  rq_init_comm_if_connected(9, "1")
  rq_init_comm_if_connected(2, "2")
  rq_init_comm_if_connected(3, "3")
  rq_init_comm_if_connected(4, "4")
  rq_print_connected_grippers()
  rq_gripper_communication_thread = run rq_gripper_communication()
  set_closed_norm(100.0, 1)
  set_open_norm(0.0, 1)
  set_closed_mm(0.0, 1)
  set_open_mm(50.0, 1)
  set_closed_norm(89.80392156862744, 2)
  set_open_norm(1.1764705882352942, 2)
  set_closed_mm(0.0, 2)
  set_open_mm(85.0, 2)
  set_closed_norm(100.0, 3)
  set_open_norm(0.0, 3)
  set_closed_mm(0.0, 3)
  set_open_mm(50.0, 3)
  set_closed_norm(100.0, 4)
  set_open_norm(0.0, 4)
  set_closed_mm(0.0, 4)
  set_open_mm(50.0, 4)
  rq_current_limit_enabled = False
  while(not rq_gripper_communication_thread_started):
      sleep(0.008)
  end
  # end: URCap Installation Node
  step_count_4a6500cf_8076_4a8b_917a_8f51ecf751d7 = 0.0
  thread Step_Counter_Thread_413bcd2b_4cc3_4dfb_b837_23a851721193():
    while (True):
      step_count_4a6500cf_8076_4a8b_917a_8f51ecf751d7 = step_count_4a6500cf_8076_4a8b_917a_8f51ecf751d7 + 1.0
      sync()
    end
  end
  run Step_Counter_Thread_413bcd2b_4cc3_4dfb_b837_23a851721193()
  global Waypoint_2_p=p[.280607659900, -.116080070486, .398046390840, -2.237106331319, 2.146374778909, -.035913347281]
  global Waypoint_2_q=[0.051861584186553955, -1.5388997805169602, -1.1589003801345825, 4.315436525935791, 1.571950912475586, 0.011884484440088272]
  global Waypoint_64_p=p[.354470099489, -.115863572825, .377183440885, -3.127244589782, -.024157028155, -.017479675085]
  global Waypoint_64_q=[0.04108531400561333, -1.8477684460081996, -0.895115852355957, 4.326324625606201, 1.5751920938491821, -1.5445211569415491]
  global Waypoint_65_p=p[.360926107403, -.115109045274, .191361701352, -3.127293402598, -.024210541102, -.017289759710]
  global Waypoint_65_q=[0.04325436055660248, -1.9099999866881312, -1.7111023664474487, 5.204389768629827, 1.5756800174713135, -1.549448315297262]
  global Waypoint_66_p=p[.360932787725, -.115104634702, .343669410000, -3.127285727102, -.024216683853, -.017394975926]
  global Waypoint_66_q=[0.042698003351688385, -1.8273731670775355, -1.0869383811950684, 4.497707052821777, 1.5746601819992065, -1.5442584196673792]
  global Waypoint_67_p=p[.360931648608, -.115099983374, .343682798901, .037017771719, -3.130286849386, .022250894461]
  global Waypoint_67_q=[0.049796681851148605, -1.8348614178099574, -1.0676213502883911, 4.462740107173584, 1.5471274852752686, 1.5965529680252075]
  global Waypoint_68_p=p[.369452922664, -.269494866094, .114409751435, .034594999463, -2.558735015916, -1.790314713905]
  global Waypoint_68_q=[-0.506531063710348, -3.1360022030272425, 0.2904461065875452, 3.4742390352436523, 2.5075576305389404, 0.5356799960136414]
  global Waypoint_79_p=p[.369461792411, -.269489790217, .091378168109, .034671000925, -2.558784123149, -1.790337845898]
  global Waypoint_79_q=[-0.5066073576556605, -3.2201863727965296, 0.36221200624574834, 3.4865333276936035, 2.507685422897339, 0.5354438424110413]
  global Waypoint_73_p=p[.355312960958, -.120113755208, .193383739669, -2.219409439704, 2.165038969222, -.036333231459]
  global Waypoint_73_q=[0.030303990468382835, -1.8856717548766078, -1.7507002353668213, 5.25380157211379, 1.5736638307571411, -0.0011132399188440445]
  global Waypoint_77_p=p[.355960533253, -.120111757755, .194005001047, -3.095268771574, .046175877951, .006344872093]
  global Waypoint_77_q=[0.02114737220108509, -1.8991791210570277, -1.7065989971160889, 5.174873578339376, 1.6078295707702637, -1.5260933081256312]
  global Waypoint_70_p=p[.369313361026, -.121750279780, .239195417816, .036983595410, -3.130201769342, .022288106508]
  global Waypoint_70_q=[0.030927900224924088, -1.8825870953001917, -1.4988759756088257, 4.941975313216009, 1.5469911098480225, 1.5737316608428955]
  global Waypoint_71_p=p[.355771906615, -.117714048296, .191403478305, -2.239338673519, 2.148294993320, -.040719651885]
  global Waypoint_71_q=[0.03811154514551163, -1.8879105053343714, -1.758138656616211, 5.26347969749526, 1.5698184967041016, -0.010163132344381154]
  global Waypoint_72_p=p[.361680845210, -.117399576394, .187815914645, -3.134574229139, .018986447884, .007833898805]
  global Waypoint_72_q=[0.038440003991127014, -1.9243623218932093, -1.7018784284591675, 5.193334001093664, 1.569042444229126, -1.5266807715045374]
  global Waypoint_75_p=p[.361669157885, -.117405189295, .336567976331, -3.134554026129, .018916398175, .007773225074]
  global Waypoint_75_q=[0.03786372393369675, -1.8343554935851039, -1.105195164680481, 4.50668923437085, 1.5680339336395264, -1.5216921011554163]
  global Waypoint_76_p=p[.369461443324, -.267242268416, .139990265830, -1.905707976787, .019547548118, .054785252250]
  global Waypoint_76_q=[-0.5030587355243128, -2.9809848270811976, 0.07564908662904912, 3.5141541200825195, 2.516566038131714, -2.5729287306415003]
  global Waypoint_78_p=p[.363433709975, -.271007124876, .085521034428, -1.833243928261, .011816409372, .027475621175]
  global Waypoint_78_q=[-0.5206573645221155, -3.1302629909911097, 0.13170367876161748, 3.4938294130512695, 2.5485825538635254, -2.691174332295553]
  global Waypoint_74_p=p[.354955148094, -.112489845695, .193442052840, -.170335331910, 3.121840961438, -.070471601362]
  global Waypoint_74_q=[0.06705623120069504, -1.8727036915221156, -1.7540733814239502, 5.212656187802114, 1.5166053771972656, 1.5219447612762451]
  global Waypoint_8_p=p[.360358944520, -.116083441389, .194376541524, -2.248047450183, 2.157812796511, .002217808263]
  global Waypoint_8_q=[0.039292335510253906, -1.9029251537718714, -1.7079429626464844, 5.199970382242956, 1.5806336402893066, -0.007966343556539357]
  global Waypoint_11_p=p[.360346612111, -.116074708299, .194372829697, -.134360355414, 3.119145978590, -.025737827061]
  global Waypoint_11_q=[0.048485033214092255, -1.8981090984740199, -1.7157262563705444, 5.205127703934469, 1.5453232526779175, 1.5264861583709717]
  global Waypoint_13_p=p[.360128512254, -.115917649696, .194944831011, -2.245984467664, 2.155060370290, -.017546589543]
  global Waypoint_13_q=[0.041585683822631836, -1.8980418644347132, -1.716995120048523, 5.215424525528707, 1.5738275051116943, -0.006153885518209279]
  global Waypoint_12_p=p[.360146406837, -.115908484738, .194960409380, -3.112369099282, -.068557507067, .019286775543]
  global Waypoint_12_q=[0.03719525411725044, -1.907412668267721, -1.6854465007781982, 5.152547257929601, 1.5902478694915771, -1.583886448537008]
  global Waypoint_14_p=p[.365368782725, -.113055548392, .194065158575, -2.254756102503, 2.163756251815, .001000413874]
  global Waypoint_14_q=[0.048927538096904755, -1.9188252888121546, -1.6842378377914429, 5.186415302544393, 1.5737271308898926, 0.0014259815216064453]
  global Waypoint_15_p=p[.365366593966, -.113055726856, .313338506786, -2.254649094383, 2.163740256071, .001003954948]
  global Waypoint_15_q=[0.04848504066467285, -1.8237744770445765, -1.2354748249053955, 4.642688437099121, 1.572627305984497, 0.005483102984726429]
  global Waypoint_23_p=p[.365372287050, -.113060920253, .392746291245, -3.129916090772, .002408869415, .018908326558]
  global Waypoint_23_q=[0.04779151454567909, -1.957900186578268, -0.647434651851654, 4.165631933803223, 1.5744084119796753, -1.519916836415426]
  global Waypoint_16_p=p[.363125696366, -.264930337535, .106644692126, -1.930464727729, -.006616513493, -.014136172145]
  global Waypoint_16_q=[-0.5062182585345667, -2.7471419773497523, -0.5786928534507751, 3.9979278284260253, 2.5275027751922607, -2.5754240194903772]
  global Waypoint_17_p=p[.359006490406, -.116088333119, .193010890574, -2.237057782096, 2.146370407089, -.035922785381]
  global Waypoint_17_q=[0.041281212121248245, -1.8952018223204554, -1.7393155097961426, 5.252011346607961, 1.5739600658416748, -0.00670034090151006]
  global Waypoint_18_p=p[.359004234930, -.116091493614, .368940192177, -2.237123790240, 2.146381621509, -.035885413675]
  global Waypoint_18_q=[0.04060101509094238, -1.8347741566100062, -0.9686561226844788, 4.42090289175, 1.5729669332504272, -7.427374469202164E-4]
  global Waypoint_19_p=p[.359011315786, -.116090988468, .368946186542, -3.094932517113, -.087303060908, .020290804464]
  global Waypoint_19_q=[0.031704679131507874, -1.8744904003539027, -0.8905159831047058, 4.323864622707031, 1.6067882776260376, -1.5951746145831507]
  global Waypoint_20_p=p[.366236911694, -.120423048900, .235895888638, -3.094888190076, -.087401744852, .020371246681]
  global Waypoint_20_q=[0.01979127898812294, -1.8803430996336878, -1.5173594951629639, 4.955764177232542, 1.6063188314437866, -1.6122682730304163]
  global Waypoint_21_p=p[.364127453615, -.117777467803, .193292956992, -2.256931465612, 2.166078680800, .016499453347]
  global Waypoint_21_q=[0.03465377166867256, -1.9235106907286585, -1.6773513555526733, 5.174797373801031, 1.5786932706832886, -0.01269084612001592]
  global Waypoint_32_p=p[.364117039848, -.117791711540, .193288967422, -.001509992748, 3.124739503024, -.003616906989]
  global Waypoint_32_q=[0.03972397744655609, -1.9184686146178187, -1.6911675930023193, 5.198225903301992, 1.558967113494873, 1.6030347347259521]
  global Waypoint_24_p=p[.356858385198, -.114748285525, .193459227445, -2.236998775234, 2.146447506006, -.035874401211]
  global Waypoint_24_q=[0.045367274433374405, -1.8846894703307093, -1.7517141103744507, 5.253918099194326, 1.5737637281417847, -0.0025556723224084976]
  global Waypoint_25_p=p[.356855401252, -.114737739719, .388234546256, -2.237156328648, 2.146401722995, -.035868096178]
  global Waypoint_25_q=[0.04460291564464569, -1.8599993191161097, -0.837320864200592, 4.314809961909912, 1.5731350183486938, 0.004033051431179047]
  global Waypoint_27_p=p[.356862717244, -.114749303796, .388207810464, -3.101225685288, -.061188193992, .021131354318]
  global Waypoint_27_q=[0.0369672067463398, -1.9050165615477503, -0.7486847043037415, 4.212594671840332, 1.6017820835113525, -1.5721553007708948]
  global Waypoint_26_p=p[.365655111079, -.272422037322, .090212739427, -1.849444862553, -.046251879190, -.014050237907]
  global Waypoint_26_q=[-0.519848648701803, -3.0603820286192835, 0.005677525197164357, 3.5761772829243164, 2.5399975776672363, -2.73091704050173]
  global Waypoint_28_p=p[.354352026237, -.116082337067, .201505476102, -2.237022096588, 2.146441145418, -.035930660985]
  global Waypoint_28_q=[0.04179730266332626, -1.861342569390768, -1.741385579109192, 5.2202181098754785, 1.573683500289917, -0.005864922200338185]
  global Waypoint_29_p=p[.354342109747, -.116082273200, .351046674865, -2.237104102966, 2.146365455752, -.035900070297]
  global Waypoint_29_q=[0.04126540571451187, -1.7894679508604945, -1.1141570806503296, 4.521125956172607, 1.5726195573806763, -8.066336261194351E-4]
  global Waypoint_30_p=p[.354353116406, -.116080119546, .351018725794, -3.094806654881, -.093017323019, .020491730000]
  global Waypoint_30_q=[0.032280921936035156, -1.824392934838766, -1.0455470085144043, 4.428581400508545, 1.6063028573989868, -1.5990260283099573]
  global Waypoint_31_p=p[.368984100378, -.120915937945, .229682487256, -3.095748275296, .014195489245, .018015526971]
  global Waypoint_31_q=[0.018162259832024574, -1.8980938396849574, -1.5245105028152466, 4.9836007235343835, 1.6071596145629883, -1.5484493414508265]
  global Waypoint_22_p=p[.364116883869, -.117782716197, .193288229298, -3.139205010194, -.012449845557, .026525647038]
  global Waypoint_22_q=[0.03819990158081055, -1.9253126583495082, -1.6663216352462769, 5.146627026587286, 1.5645008087158203, -1.5466154257403772]
  global Waypoint_33_p=p[.365384650811, -.113046739845, .368046327177, -.082065141775, 3.127997038214, -.017202640169]
  global Waypoint_33_q=[0.05418265983462334, -1.8752075634398402, -0.9042851328849792, 4.363438292140625, 1.5500004291534424, 1.5726572275161743]
  global Waypoint_34_p=p[.363742157567, -.276249559590, .088704299793, -.017752167727, 2.507683090614, 1.878743902822]
  global Waypoint_34_q=[-0.5293481985675257, -3.0111896000304164, -0.10669158399105072, 3.651848478908203, 2.5413897037506104, 0.4435216784477234]
  global Waypoint_35_p=p[.365353984843, -.113065797339, .314962777279, -3.129998929491, -.008745881210, .018959456628]
  global Waypoint_35_q=[0.04835740104317665, -1.834442754785055, -1.204733967781067, 4.599378271693848, 1.5727750062942505, -1.5296428839312952]
  global Waypoint_36_p=p[.365363249284, -.113054207165, .238209290372, -3.129975666367, -.008814066519, .018790901880]
  global Waypoint_36_q=[0.04866836220026016, -1.8599559269347132, -1.5340592861175537, 4.954310434847631, 1.573059320449829, -1.532309357319967]
  global Waypoint_37_p=p[.365360195551, -.113055658309, .193805528531, -3.129976498904, -.008769838028, .018833791209]
  global Waypoint_37_q=[0.04882422462105751, -1.923554082910055, -1.6685000658035278, 5.152311789780416, 1.573791742324829, -1.5337484518634241]
  global Waypoint_38_p=p[.364249601416, -.113557103657, .190832473293, 2.204318959610, 2.224300240519, -.048856099106]
  global Waypoint_38_q=[0.05790204554796219, -1.921460290948385, -1.6850007772445679, 5.161710727005758, 1.5336676836013794, -3.0986831823932093]
  global Waypoint_39_p=p[.364266614325, -.110421946332, .190856746275, 2.209420651831, 2.229591677071, -.037414170316]
  global Waypoint_39_q=[0.06399016082286835, -1.9190217457213343, -1.6884911060333252, 5.163263070374288, 1.544034719467163, -3.092748228703634]
  global Waypoint_40_p=p[.364268983895, -.110435285300, .361886964377, 2.209420466399, 2.229618306717, -.037429530523]
  global Waypoint_40_q=[0.06325225532054901, -1.8707810841002406, -0.9290131330490112, 4.355386896724365, 1.5435824394226074, -3.086977783833639]
  global Waypoint_41_p=p[.364265840443, -.110427102269, .361870025237, -3.125110448973, -.105776433446, .029932400516]
  global Waypoint_41_q=[0.05484846606850624, -1.8776551685728968, -0.9186587929725647, 4.349270983333252, 1.5762443542480469, -1.5833638350116175]
  global Waypoint_42_p=p[.369042632900, -.110424594122, .224326920210, -3.126301319343, -.005632380127, .029185961145]
  global Waypoint_42_q=[0.05444587022066116, -1.889749666253561, -1.5589039325714111, 5.0025426028068445, 1.5772563219070435, -1.5249899069415491]
  global Waypoint_43_p=p[.365353936489, -.113064268181, .322294641646, -2.254796238667, 2.163800975117, .001120761204]
  global Waypoint_43_q=[0.04843675345182419, -1.8276883564391078, -1.1881848573684692, 4.59915463506665, 1.5726237297058105, 0.0057464404962956905]
  global Waypoint_44_p=p[.365369713945, -.113043464009, .322292976272, -3.129186148249, -.086620865562, .019272676305]
  global Waypoint_44_q=[0.04855327680706978, -1.8383614025511683, -1.1648505926132202, 4.562915487880371, 1.5721629858016968, -1.5789158979998987]
  global Waypoint_45_p=p[.365392044628, -.271165795022, .097080861471, -1.854532438468, -.060032954149, -.026643104538]
  global Waypoint_45_q=[-0.5176385084735315, -2.9681459865965785, -0.158863827586174, 3.659778280849121, 2.540245294570923, -2.7370362917529505]
  global Waypoint_46_p=p[.365359176267, -.113063290570, .333428241271, -2.254692977086, 2.163738544463, .000970293766]
  global Waypoint_46_q=[0.04838533699512482, -1.8350216350951136, -1.1259797811508179, 4.544436617488525, 1.5727194547653198, 0.006145970430225134]
  global Waypoint_47_p=p[.365371307895, -.113054913652, .333395021784, -3.130121874518, -.066020013586, .019874548846]
  global Waypoint_47_q=[0.048556797206401825, -1.8465644321837367, -1.1012637615203857, 4.507215185756348, 1.5719189643859863, -1.565303150807516]
  global Waypoint_48_p=p[.365368433594, -.110775889601, .232224413161, -3.130138965271, -.066016593977, .019854438479]
  global Waypoint_48_q=[0.0552668571472168, -1.8638464413084925, -1.5576152801513672, 4.98091487863616, 1.5721588134765625, -1.562469784413473]
  global Waypoint_52_p=p[.365359843959, -.113081349965, .194064897071, -3.129642378612, -.064303807651, .019061278977]
  global Waypoint_52_q=[0.04888356477022171, -1.9231182537474574, -1.667611002922058, 5.150625216751852, 1.5732671022415161, -1.5691588560687464]
  global Waypoint_49_p=p[.365357344058, -.113073281521, .368518599816, -3.129675426161, -.064295774517, .019011934194]
  global Waypoint_49_q=[0.04817046970129013, -1.8945962391295375, -0.8649749755859375, 4.319530649776123, 1.5729867219924927, -1.5631969610797327]
  global Waypoint_50_p=p[.371009155844, -.266422439514, .106051816126, -1.904984487247, -.030855415702, .036523254658]
  global Waypoint_50_q=[-0.49856454530824834, -2.904177804986471, -0.24639520049095154, 3.7509915071674804, 2.5077571868896484, -2.622943703328268]
  global Waypoint_51_p=p[.365365756281, -.113068067212, .335109436071, -2.254715734372, 2.163808014871, .001013615422]
  global Waypoint_51_q=[0.048369091004133224, -1.8364578686156214, -1.116073727607727, 4.535901232356689, 1.5727112293243408, 0.0062180995009839535]
  global Waypoint_53_p=p[.363190347376, -.109909249167, .214454177245, 2.202648627526, 2.239361144151, -.026164233321]
  global Waypoint_53_q=[0.0639103502035141, -1.8745748005309046, -1.631171464920044, 5.0654775378997705, 1.5498764514923096, -3.099539581929342]
  global Waypoint_54_p=p[.365364617238, -.113046544047, .193803919468, -2.147317235435, 2.270276089319, -.000280218377]
  global Waypoint_54_q=[0.04924694821238518, -1.9189378223814906, -1.6859766244888306, 5.189448195486822, 1.572607398033142, 0.0985577404499054]
  global Waypoint_55_p=p[.369046237243, -.110420112971, .224327646614, -2.257586529246, 2.150383646731, .005568399145]
  global Waypoint_55_q=[0.05381538346409798, -1.8819652996458949, -1.5833349227905273, 5.051859217673101, 1.5802409648895264, 4.339217866800027E-6]
  global Waypoint_56_p=p[.364264927128, -.116054024615, .192333636877, -3.095046149511, .058807189831, .016907900219]
  global Waypoint_56_q=[0.03184909746050835, -1.929457803765768, -1.669385313987732, 5.161799806147375, 1.6082003116607666, -1.5073078314410608]
  global Waypoint_57_p=p[.364253565471, -.116069606295, .333900611097, -3.095734687662, -.040512408598, .019114780625]
  global Waypoint_57_q=[0.031436286866664886, -1.85087313274526, -1.0939775705337524, 4.505091353053711, 1.6066334247589111, -1.5665701071368616]
  global Waypoint_58_p=p[.365317983006, -.268384127780, .096470187856, -1.827396022314, -.032757791678, -.006341395965]
  global Waypoint_58_q=[-0.514263931904928, -3.06442989925527, 0.04053718248476201, 3.5144497591206054, 2.5557875633239746, -2.7419408003436487]
  global Waypoint_59_p=p[.361348202281, -.116091074418, .193171940183, -2.255348123474, 2.164443027209, .005235593744]
  global Waypoint_59_q=[0.04056864231824875, -1.9096676311888636, -1.7008389234542847, 5.191219466715612, 1.5751317739486694, -0.006904427205220998]
  global Waypoint_60_p=p[.361353719735, -.116078329177, .193164234402, -.107411230804, 3.126172424726, -.013320009558]
  global Waypoint_60_q=[0.04628801345825195, -1.906170507470602, -1.7079107761383057, 5.199406075268545, 1.553221583366394, 1.5418486595153809]
  global Waypoint_62_p=p[.357407157421, -.114500090328, .192443539627, -2.237115183190, 2.146339057492, -.035930597557]
  global Waypoint_62_q=[0.04602402448654175, -1.8884631596007289, -1.7518619298934937, 5.257864701538839, 1.5737314224243164, -0.0020354429828088882]
  global Waypoint_61_p=p[.357808555570, -.114512094935, .192817914002, -3.094022297870, -.120534455071, .014031671817]
  global Waypoint_61_q=[0.037067364901304245, -1.9025441608824671, -1.7050750255584717, 5.170009690314092, 1.6068851947784424, -1.6179912726031702]
  global Waypoint_63_p=p[.361345425225, -.116096314852, .193167637645, 2.081805564531, 2.284545736471, .059854815242]
  global Waypoint_63_q=[0.04617943987250328, -1.8987189731993617, -1.7417824268341064, 5.275271165161886, 1.5542293787002563, 3.087625741958618]
  $ 2 "Robot Program"
  $ 3 "Mouvements L'"
  $ 4 "MoveJ"
  $ 5 "Waypoint_2" "breakAfter"
  movej(get_inverse_kin(Waypoint_2_p, qnear=Waypoint_2_q), a=1.3962634015954636, v=1.0471975511965976)
  $ 6 "MoveJ"
  $ 7 "Waypoint_64" "breakAfter"
  movej(get_inverse_kin(Waypoint_64_p, qnear=Waypoint_64_q), a=1.3962634015954636, v=1.0471975511965976)
  $ 8 "MoveJ"
  $ 9 "Waypoint_65" "breakAfter"
  movej(get_inverse_kin(Waypoint_65_p, qnear=Waypoint_65_q), a=1.3962634015954636, v=1.0471975511965976)
  # begin: URCap Program Node
  #   Source: Robotiq_Grippers, 1.8.11.21258, Robotiq Inc.
  #   Type: Gripper
  $ 10 "Gripper Close (2)"
  if not(gripper_connected[1]):
    popup("Gripper 2 must be connected to run this program.", "No connection", False, True, True)
  end
  if not(rq_is_gripper_activated("2")):
    popup("Gripper 2 is not activated. Go to Installation tab > Gripper to activate it and run the program again.", "Not activated", False, True, True)
  end
  rq_set_pos_spd_for(255, 0, 0, "2")
  rq_wait_pos_spe_for_request(255, 0, 0, "2")
  rq_go_to("2")
  rq_wait("2")
  # end: URCap Program Node
  $ 11 "MoveJ"
  $ 12 "Waypoint_66" "breakAfter"
  movej(get_inverse_kin(Waypoint_66_p, qnear=Waypoint_66_q), a=1.3962634015954636, v=1.0471975511965976)
  $ 13 "MoveJ"
  $ 14 "Waypoint_67" "breakAfter"
  movej(get_inverse_kin(Waypoint_67_p, qnear=Waypoint_67_q), a=1.3962634015954636, v=1.0471975511965976)
  $ 15 "MoveJ"
  $ 16 "Waypoint_68" "breakAfter"
  movej(get_inverse_kin(Waypoint_68_p, qnear=Waypoint_68_q), a=1.3962634015954636, v=1.0471975511965976)
  $ 17 "MoveJ"
  $ 18 "Waypoint_79" "breakAfter"
  movej(get_inverse_kin(Waypoint_79_p, qnear=Waypoint_79_q), a=1.3962634015954636, v=1.0471975511965976)
  # begin: URCap Program Node
  #   Source: Robotiq_Grippers, 1.8.11.21258, Robotiq Inc.
  #   Type: Gripper
  $ 19 "Gripper Open (2)"
  if not(gripper_connected[1]):
    popup("Gripper 2 must be connected to run this program.", "No connection", False, True, True)
  end
  if not(rq_is_gripper_activated("2")):
    popup("Gripper 2 is not activated. Go to Installation tab > Gripper to activate it and run the program again.", "Not activated", False, True, True)
  end
  rq_set_pos_spd_for(0, 0, 0, "2")
  rq_wait_pos_spe_for_request(0, 0, 0, "2")
  rq_go_to("2")
  rq_wait("2")
  # end: URCap Program Node
  $ 20 "MoveJ"
  $ 21 "Waypoint_2" "breakAfter"
  movej(get_inverse_kin(Waypoint_2_p, qnear=Waypoint_2_q), a=1.3962634015954636, v=1.0471975511965976)
  $ 22 "MoveJ"
  $ 23 "MoveJ"
  $ 24 "MoveJ"
  $ 25 "MoveJ"
  $ 26 "MoveJ"
  $ 27 "MoveJ"
  $ 28 "Waypoint_73" "breakAfter"
  movej(get_inverse_kin(Waypoint_73_p, qnear=Waypoint_73_q), a=1.3962634015954636, v=1.0471975511965976)
  # begin: URCap Program Node
  #   Source: Robotiq_Grippers, 1.8.11.21258, Robotiq Inc.
  #   Type: Gripper
  $ 29 "Gripper Close (2)"
  if not(gripper_connected[1]):
    popup("Gripper 2 must be connected to run this program.", "No connection", False, True, True)
  end
  if not(rq_is_gripper_activated("2")):
    popup("Gripper 2 is not activated. Go to Installation tab > Gripper to activate it and run the program again.", "Not activated", False, True, True)
  end
  rq_set_pos_spd_for(255, 0, 0, "2")
  rq_wait_pos_spe_for_request(255, 0, 0, "2")
  rq_go_to("2")
  rq_wait("2")
  # end: URCap Program Node
  $ 30 "MoveJ"
  $ 31 "Waypoint_77" "breakAfter"
  movej(get_inverse_kin(Waypoint_77_p, qnear=Waypoint_77_q), a=1.3962634015954636, v=1.0471975511965976)
  # begin: URCap Program Node
  #   Source: Robotiq_Grippers, 1.8.11.21258, Robotiq Inc.
  #   Type: Gripper
  $ 32 "Gripper Open (2)"
  if not(gripper_connected[1]):
    popup("Gripper 2 must be connected to run this program.", "No connection", False, True, True)
  end
  if not(rq_is_gripper_activated("2")):
    popup("Gripper 2 is not activated. Go to Installation tab > Gripper to activate it and run the program again.", "Not activated", False, True, True)
  end
  rq_set_pos_spd_for(0, 0, 0, "2")
  rq_wait_pos_spe_for_request(0, 0, 0, "2")
  rq_go_to("2")
  rq_wait("2")
  # end: URCap Program Node
  $ 33 "MoveJ"
  $ 34 "Waypoint_2" "breakAfter"
  movej(get_inverse_kin(Waypoint_2_p, qnear=Waypoint_2_q), a=1.3962634015954636, v=1.0471975511965976)
  $ 35 "MoveJ"
  $ 36 "Waypoint_64" "breakAfter"
  movej(get_inverse_kin(Waypoint_64_p, qnear=Waypoint_64_q), a=1.3962634015954636, v=1.0471975511965976)
  $ 37 "MoveJ"
  $ 38 "Waypoint_65" "breakAfter"
  movej(get_inverse_kin(Waypoint_65_p, qnear=Waypoint_65_q), a=1.3962634015954636, v=1.0471975511965976)
  # begin: URCap Program Node
  #   Source: Robotiq_Grippers, 1.8.11.21258, Robotiq Inc.
  #   Type: Gripper
  $ 39 "Gripper Close (2)"
  if not(gripper_connected[1]):
    popup("Gripper 2 must be connected to run this program.", "No connection", False, True, True)
  end
  if not(rq_is_gripper_activated("2")):
    popup("Gripper 2 is not activated. Go to Installation tab > Gripper to activate it and run the program again.", "Not activated", False, True, True)
  end
  rq_set_pos_spd_for(255, 0, 0, "2")
  rq_wait_pos_spe_for_request(255, 0, 0, "2")
  rq_go_to("2")
  rq_wait("2")
  # end: URCap Program Node
  $ 40 "MoveJ"
  $ 41 "Waypoint_66" "breakAfter"
  movej(get_inverse_kin(Waypoint_66_p, qnear=Waypoint_66_q), a=1.3962634015954636, v=1.0471975511965976)
  $ 42 "MoveJ"
  $ 43 "Waypoint_67" "breakAfter"
  movej(get_inverse_kin(Waypoint_67_p, qnear=Waypoint_67_q), a=1.3962634015954636, v=1.0471975511965976)
  $ 44 "MoveJ"
  $ 45 "Waypoint_70" "breakAfter"
  movej(get_inverse_kin(Waypoint_70_p, qnear=Waypoint_70_q), a=1.3962634015954636, v=1.0471975511965976)
  # begin: URCap Program Node
  #   Source: Robotiq_Grippers, 1.8.11.21258, Robotiq Inc.
  #   Type: Gripper
  $ 46 "Gripper Open (2)"
  if not(gripper_connected[1]):
    popup("Gripper 2 must be connected to run this program.", "No connection", False, True, True)
  end
  if not(rq_is_gripper_activated("2")):
    popup("Gripper 2 is not activated. Go to Installation tab > Gripper to activate it and run the program again.", "Not activated", False, True, True)
  end
  rq_set_pos_spd_for(0, 0, 0, "2")
  rq_wait_pos_spe_for_request(0, 0, 0, "2")
  rq_go_to("2")
  rq_wait("2")
  # end: URCap Program Node
  $ 47 "MoveJ"
  $ 48 "Waypoint_2" "breakAfter"
  movej(get_inverse_kin(Waypoint_2_p, qnear=Waypoint_2_q), a=1.3962634015954636, v=1.0471975511965976)
  $ 49 "MoveJ"
  $ 50 "Waypoint_71" "breakAfter"
  movej(get_inverse_kin(Waypoint_71_p, qnear=Waypoint_71_q), a=1.3962634015954636, v=1.0471975511965976)
  # begin: URCap Program Node
  #   Source: Robotiq_Grippers, 1.8.11.21258, Robotiq Inc.
  #   Type: Gripper
  $ 51 "Gripper Close (2)"
  if not(gripper_connected[1]):
    popup("Gripper 2 must be connected to run this program.", "No connection", False, True, True)
  end
  if not(rq_is_gripper_activated("2")):
    popup("Gripper 2 is not activated. Go to Installation tab > Gripper to activate it and run the program again.", "Not activated", False, True, True)
  end
  rq_set_pos_spd_for(255, 0, 0, "2")
  rq_wait_pos_spe_for_request(255, 0, 0, "2")
  rq_go_to("2")
  rq_wait("2")
  # end: URCap Program Node
  # begin: URCap Program Node
  #   Source: Robotiq_Grippers, 1.8.11.21258, Robotiq Inc.
  #   Type: Gripper
  $ 52 "Gripper Open (2)"
  if not(gripper_connected[1]):
    popup("Gripper 2 must be connected to run this program.", "No connection", False, True, True)
  end
  if not(rq_is_gripper_activated("2")):
    popup("Gripper 2 is not activated. Go to Installation tab > Gripper to activate it and run the program again.", "Not activated", False, True, True)
  end
  rq_set_pos_spd_for(0, 0, 0, "2")
  rq_wait_pos_spe_for_request(0, 0, 0, "2")
  rq_go_to("2")
  rq_wait("2")
  # end: URCap Program Node
  $ 53 "MoveJ"
  $ 54 "Waypoint_72" "breakAfter"
  movej(get_inverse_kin(Waypoint_72_p, qnear=Waypoint_72_q), a=1.3962634015954636, v=1.0471975511965976)
  # begin: URCap Program Node
  #   Source: Robotiq_Grippers, 1.8.11.21258, Robotiq Inc.
  #   Type: Gripper
  $ 55 "Gripper Close (2)"
  if not(gripper_connected[1]):
    popup("Gripper 2 must be connected to run this program.", "No connection", False, True, True)
  end
  if not(rq_is_gripper_activated("2")):
    popup("Gripper 2 is not activated. Go to Installation tab > Gripper to activate it and run the program again.", "Not activated", False, True, True)
  end
  rq_set_pos_spd_for(255, 0, 0, "2")
  rq_wait_pos_spe_for_request(255, 0, 0, "2")
  rq_go_to("2")
  rq_wait("2")
  # end: URCap Program Node
  $ 56 "MoveJ"
  $ 57 "Waypoint_75" "breakAfter"
  movej(get_inverse_kin(Waypoint_75_p, qnear=Waypoint_75_q), a=1.3962634015954636, v=1.0471975511965976)
  $ 58 "MoveJ"
  $ 59 "Waypoint_76" "breakAfter"
  movej(get_inverse_kin(Waypoint_76_p, qnear=Waypoint_76_q), a=1.3962634015954636, v=1.0471975511965976)
  $ 60 "MoveJ"
  $ 61 "Waypoint_78" "breakAfter"
  movej(get_inverse_kin(Waypoint_78_p, qnear=Waypoint_78_q), a=1.3962634015954636, v=1.0471975511965976)
  $ 62 "Waypoint_78" "breakAfter"
  movej(get_inverse_kin(Waypoint_78_p, qnear=Waypoint_78_q), a=1.3962634015954636, v=1.0471975511965976)
  # begin: URCap Program Node
  #   Source: Robotiq_Grippers, 1.8.11.21258, Robotiq Inc.
  #   Type: Gripper
  $ 63 "Gripper Open (2)"
  if not(gripper_connected[1]):
    popup("Gripper 2 must be connected to run this program.", "No connection", False, True, True)
  end
  if not(rq_is_gripper_activated("2")):
    popup("Gripper 2 is not activated. Go to Installation tab > Gripper to activate it and run the program again.", "Not activated", False, True, True)
  end
  rq_set_pos_spd_for(0, 0, 0, "2")
  rq_wait_pos_spe_for_request(0, 0, 0, "2")
  rq_go_to("2")
  rq_wait("2")
  # end: URCap Program Node
  $ 64 "MoveJ"
  $ 65 "Waypoint_2" "breakAfter"
  movej(get_inverse_kin(Waypoint_2_p, qnear=Waypoint_2_q), a=1.3962634015954636, v=1.0471975511965976)
  $ 66 "Mouvements L"
  $ 67 "MoveJ"
  $ 68 "Waypoint_2" "breakAfter"
  movej(get_inverse_kin(Waypoint_2_p, qnear=Waypoint_2_q), a=1.3962634015954636, v=1.0471975511965976)
  $ 69 "MoveJ"
  $ 70 "Waypoint_64" "breakAfter"
  movej(get_inverse_kin(Waypoint_64_p, qnear=Waypoint_64_q), a=1.3962634015954636, v=1.0471975511965976)
  $ 71 "MoveJ"
  $ 72 "Waypoint_65" "breakAfter"
  movej(get_inverse_kin(Waypoint_65_p, qnear=Waypoint_65_q), a=1.3962634015954636, v=1.0471975511965976)
  # begin: URCap Program Node
  #   Source: Robotiq_Grippers, 1.8.11.21258, Robotiq Inc.
  #   Type: Gripper
  $ 73 "Gripper Close (2)"
  if not(gripper_connected[1]):
    popup("Gripper 2 must be connected to run this program.", "No connection", False, True, True)
  end
  if not(rq_is_gripper_activated("2")):
    popup("Gripper 2 is not activated. Go to Installation tab > Gripper to activate it and run the program again.", "Not activated", False, True, True)
  end
  rq_set_pos_spd_for(255, 0, 0, "2")
  rq_wait_pos_spe_for_request(255, 0, 0, "2")
  rq_go_to("2")
  rq_wait("2")
  # end: URCap Program Node
  $ 74 "MoveJ"
  $ 75 "Waypoint_66" "breakAfter"
  movej(get_inverse_kin(Waypoint_66_p, qnear=Waypoint_66_q), a=1.3962634015954636, v=1.0471975511965976)
  $ 76 "MoveJ"
  $ 77 "Waypoint_67" "breakAfter"
  movej(get_inverse_kin(Waypoint_67_p, qnear=Waypoint_67_q), a=1.3962634015954636, v=1.0471975511965976)
  $ 78 "MoveJ"
  $ 79 "Waypoint_68" "breakAfter"
  movej(get_inverse_kin(Waypoint_68_p, qnear=Waypoint_68_q), a=1.3962634015954636, v=1.0471975511965976)
  $ 80 "MoveJ"
  $ 81 "Waypoint_79" "breakAfter"
  movej(get_inverse_kin(Waypoint_79_p, qnear=Waypoint_79_q), a=1.3962634015954636, v=1.0471975511965976)
  # begin: URCap Program Node
  #   Source: Robotiq_Grippers, 1.8.11.21258, Robotiq Inc.
  #   Type: Gripper
  $ 82 "Gripper Open (2)"
  if not(gripper_connected[1]):
    popup("Gripper 2 must be connected to run this program.", "No connection", False, True, True)
  end
  if not(rq_is_gripper_activated("2")):
    popup("Gripper 2 is not activated. Go to Installation tab > Gripper to activate it and run the program again.", "Not activated", False, True, True)
  end
  rq_set_pos_spd_for(0, 0, 0, "2")
  rq_wait_pos_spe_for_request(0, 0, 0, "2")
  rq_go_to("2")
  rq_wait("2")
  # end: URCap Program Node
  $ 83 "MoveJ"
  $ 84 "Waypoint_2" "breakAfter"
  movej(get_inverse_kin(Waypoint_2_p, qnear=Waypoint_2_q), a=1.3962634015954636, v=1.0471975511965976)
  $ 85 "MoveJ"
  $ 86 "MoveJ"
  $ 87 "MoveJ"
  $ 88 "MoveJ"
  $ 89 "MoveJ"
  $ 90 "Waypoint_2" "breakAfter"
  movej(get_inverse_kin(Waypoint_2_p, qnear=Waypoint_2_q), a=1.3962634015954636, v=1.0471975511965976)
  $ 91 "MoveJ"
  $ 92 "Waypoint_73" "breakAfter"
  movej(get_inverse_kin(Waypoint_73_p, qnear=Waypoint_73_q), a=1.3962634015954636, v=1.0471975511965976)
  # begin: URCap Program Node
  #   Source: Robotiq_Grippers, 1.8.11.21258, Robotiq Inc.
  #   Type: Gripper
  $ 93 "Gripper Close (2)"
  if not(gripper_connected[1]):
    popup("Gripper 2 must be connected to run this program.", "No connection", False, True, True)
  end
  if not(rq_is_gripper_activated("2")):
    popup("Gripper 2 is not activated. Go to Installation tab > Gripper to activate it and run the program again.", "Not activated", False, True, True)
  end
  rq_set_pos_spd_for(255, 0, 0, "2")
  rq_wait_pos_spe_for_request(255, 0, 0, "2")
  rq_go_to("2")
  rq_wait("2")
  # end: URCap Program Node
  $ 94 "MoveJ"
  $ 95 "Waypoint_74" "breakAfter"
  movej(get_inverse_kin(Waypoint_74_p, qnear=Waypoint_74_q), a=1.3962634015954636, v=1.0471975511965976)
  # begin: URCap Program Node
  #   Source: Robotiq_Grippers, 1.8.11.21258, Robotiq Inc.
  #   Type: Gripper
  $ 96 "Gripper Open (2)"
  if not(gripper_connected[1]):
    popup("Gripper 2 must be connected to run this program.", "No connection", False, True, True)
  end
  if not(rq_is_gripper_activated("2")):
    popup("Gripper 2 is not activated. Go to Installation tab > Gripper to activate it and run the program again.", "Not activated", False, True, True)
  end
  rq_set_pos_spd_for(0, 0, 0, "2")
  rq_wait_pos_spe_for_request(0, 0, 0, "2")
  rq_go_to("2")
  rq_wait("2")
  # end: URCap Program Node
  $ 97 "MoveJ"
  $ 98 "Waypoint_2" "breakAfter"
  movej(get_inverse_kin(Waypoint_2_p, qnear=Waypoint_2_q), a=1.3962634015954636, v=1.0471975511965976)
  $ 99 "MoveJ"
  $ 100 "Waypoint_64" "breakAfter"
  movej(get_inverse_kin(Waypoint_64_p, qnear=Waypoint_64_q), a=1.3962634015954636, v=1.0471975511965976)
  $ 101 "MoveJ"
  $ 102 "Waypoint_65" "breakAfter"
  movej(get_inverse_kin(Waypoint_65_p, qnear=Waypoint_65_q), a=1.3962634015954636, v=1.0471975511965976)
  # begin: URCap Program Node
  #   Source: Robotiq_Grippers, 1.8.11.21258, Robotiq Inc.
  #   Type: Gripper
  $ 103 "Gripper Close (2)"
  if not(gripper_connected[1]):
    popup("Gripper 2 must be connected to run this program.", "No connection", False, True, True)
  end
  if not(rq_is_gripper_activated("2")):
    popup("Gripper 2 is not activated. Go to Installation tab > Gripper to activate it and run the program again.", "Not activated", False, True, True)
  end
  rq_set_pos_spd_for(255, 0, 0, "2")
  rq_wait_pos_spe_for_request(255, 0, 0, "2")
  rq_go_to("2")
  rq_wait("2")
  # end: URCap Program Node
  $ 104 "MoveJ"
  $ 105 "Waypoint_66" "breakAfter"
  movej(get_inverse_kin(Waypoint_66_p, qnear=Waypoint_66_q), a=1.3962634015954636, v=1.0471975511965976)
  $ 106 "MoveJ"
  $ 107 "Waypoint_67" "breakAfter"
  movej(get_inverse_kin(Waypoint_67_p, qnear=Waypoint_67_q), a=1.3962634015954636, v=1.0471975511965976)
  $ 108 "MoveJ"
  $ 109 "Waypoint_70" "breakAfter"
  movej(get_inverse_kin(Waypoint_70_p, qnear=Waypoint_70_q), a=1.3962634015954636, v=1.0471975511965976)
  # begin: URCap Program Node
  #   Source: Robotiq_Grippers, 1.8.11.21258, Robotiq Inc.
  #   Type: Gripper
  $ 110 "Gripper Open (2)"
  if not(gripper_connected[1]):
    popup("Gripper 2 must be connected to run this program.", "No connection", False, True, True)
  end
  if not(rq_is_gripper_activated("2")):
    popup("Gripper 2 is not activated. Go to Installation tab > Gripper to activate it and run the program again.", "Not activated", False, True, True)
  end
  rq_set_pos_spd_for(0, 0, 0, "2")
  rq_wait_pos_spe_for_request(0, 0, 0, "2")
  rq_go_to("2")
  rq_wait("2")
  # end: URCap Program Node
  $ 111 "MoveJ"
  $ 112 "Waypoint_2" "breakAfter"
  movej(get_inverse_kin(Waypoint_2_p, qnear=Waypoint_2_q), a=1.3962634015954636, v=1.0471975511965976)
  $ 113 "MoveJ"
  $ 114 "Waypoint_71" "breakAfter"
  movej(get_inverse_kin(Waypoint_71_p, qnear=Waypoint_71_q), a=1.3962634015954636, v=1.0471975511965976)
  # begin: URCap Program Node
  #   Source: Robotiq_Grippers, 1.8.11.21258, Robotiq Inc.
  #   Type: Gripper
  $ 115 "Gripper Close (2)"
  if not(gripper_connected[1]):
    popup("Gripper 2 must be connected to run this program.", "No connection", False, True, True)
  end
  if not(rq_is_gripper_activated("2")):
    popup("Gripper 2 is not activated. Go to Installation tab > Gripper to activate it and run the program again.", "Not activated", False, True, True)
  end
  rq_set_pos_spd_for(255, 0, 0, "2")
  rq_wait_pos_spe_for_request(255, 0, 0, "2")
  rq_go_to("2")
  rq_wait("2")
  # end: URCap Program Node
  # begin: URCap Program Node
  #   Source: Robotiq_Grippers, 1.8.11.21258, Robotiq Inc.
  #   Type: Gripper
  $ 116 "Gripper Open (2)"
  if not(gripper_connected[1]):
    popup("Gripper 2 must be connected to run this program.", "No connection", False, True, True)
  end
  if not(rq_is_gripper_activated("2")):
    popup("Gripper 2 is not activated. Go to Installation tab > Gripper to activate it and run the program again.", "Not activated", False, True, True)
  end
  rq_set_pos_spd_for(0, 0, 0, "2")
  rq_wait_pos_spe_for_request(0, 0, 0, "2")
  rq_go_to("2")
  rq_wait("2")
  # end: URCap Program Node
  $ 117 "MoveJ"
  $ 118 "Waypoint_72" "breakAfter"
  movej(get_inverse_kin(Waypoint_72_p, qnear=Waypoint_72_q), a=1.3962634015954636, v=1.0471975511965976)
  # begin: URCap Program Node
  #   Source: Robotiq_Grippers, 1.8.11.21258, Robotiq Inc.
  #   Type: Gripper
  $ 119 "Gripper Close (2)"
  if not(gripper_connected[1]):
    popup("Gripper 2 must be connected to run this program.", "No connection", False, True, True)
  end
  if not(rq_is_gripper_activated("2")):
    popup("Gripper 2 is not activated. Go to Installation tab > Gripper to activate it and run the program again.", "Not activated", False, True, True)
  end
  rq_set_pos_spd_for(255, 0, 0, "2")
  rq_wait_pos_spe_for_request(255, 0, 0, "2")
  rq_go_to("2")
  rq_wait("2")
  # end: URCap Program Node
  $ 120 "MoveJ"
  $ 121 "Waypoint_75" "breakAfter"
  movej(get_inverse_kin(Waypoint_75_p, qnear=Waypoint_75_q), a=1.3962634015954636, v=1.0471975511965976)
  $ 122 "MoveJ"
  $ 123 "Waypoint_76" "breakAfter"
  movej(get_inverse_kin(Waypoint_76_p, qnear=Waypoint_76_q), a=1.3962634015954636, v=1.0471975511965976)
  $ 124 "MoveJ"
  $ 125 "Waypoint_78" "breakAfter"
  movej(get_inverse_kin(Waypoint_78_p, qnear=Waypoint_78_q), a=1.3962634015954636, v=1.0471975511965976)
  # begin: URCap Program Node
  #   Source: Robotiq_Grippers, 1.8.11.21258, Robotiq Inc.
  #   Type: Gripper
  $ 126 "Gripper Open (2)"
  if not(gripper_connected[1]):
    popup("Gripper 2 must be connected to run this program.", "No connection", False, True, True)
  end
  if not(rq_is_gripper_activated("2")):
    popup("Gripper 2 is not activated. Go to Installation tab > Gripper to activate it and run the program again.", "Not activated", False, True, True)
  end
  rq_set_pos_spd_for(0, 0, 0, "2")
  rq_wait_pos_spe_for_request(0, 0, 0, "2")
  rq_go_to("2")
  rq_wait("2")
  # end: URCap Program Node
  $ 127 "MoveJ"
  $ 128 "Waypoint_2" "breakAfter"
  movej(get_inverse_kin(Waypoint_2_p, qnear=Waypoint_2_q), a=1.3962634015954636, v=1.0471975511965976)
  $ 129 "Mouvement U"
  $ 130 "MoveJ"
  $ 131 "Waypoint_2" "breakAfter"
  movej(get_inverse_kin(Waypoint_2_p, qnear=Waypoint_2_q), a=1.3962634015954636, v=1.0471975511965976)
  $ 132 "MoveJ"
  $ 133 "Waypoint_8" "breakAfter"
  movej(get_inverse_kin(Waypoint_8_p, qnear=Waypoint_8_q), a=1.3962634015954636, v=1.0471975511965976)
  # begin: URCap Program Node
  #   Source: Robotiq_Grippers, 1.8.11.21258, Robotiq Inc.
  #   Type: Gripper
  $ 134 "Gripper Close (2)"
  if not(gripper_connected[1]):
    popup("Gripper 2 must be connected to run this program.", "No connection", False, True, True)
  end
  if not(rq_is_gripper_activated("2")):
    popup("Gripper 2 is not activated. Go to Installation tab > Gripper to activate it and run the program again.", "Not activated", False, True, True)
  end
  rq_set_pos_spd_for(255, 0, 0, "2")
  rq_wait_pos_spe_for_request(255, 0, 0, "2")
  rq_go_to("2")
  rq_wait("2")
  # end: URCap Program Node
  $ 135 "MoveJ"
  $ 136 "Waypoint_11" "breakAfter"
  movej(get_inverse_kin(Waypoint_11_p, qnear=Waypoint_11_q), a=1.3962634015954636, v=1.0471975511965976)
  # begin: URCap Program Node
  #   Source: Robotiq_Grippers, 1.8.11.21258, Robotiq Inc.
  #   Type: Gripper
  $ 137 "Gripper Open (2)"
  if not(gripper_connected[1]):
    popup("Gripper 2 must be connected to run this program.", "No connection", False, True, True)
  end
  if not(rq_is_gripper_activated("2")):
    popup("Gripper 2 is not activated. Go to Installation tab > Gripper to activate it and run the program again.", "Not activated", False, True, True)
  end
  rq_set_pos_spd_for(0, 0, 0, "2")
  rq_wait_pos_spe_for_request(0, 0, 0, "2")
  rq_go_to("2")
  rq_wait("2")
  # end: URCap Program Node
  $ 138 "MoveJ"
  $ 139 "Waypoint_2" "breakAfter"
  movej(get_inverse_kin(Waypoint_2_p, qnear=Waypoint_2_q), a=1.3962634015954636, v=1.0471975511965976)
  $ 140 "Mouvement U'"
  $ 141 "MoveJ"
  $ 142 "Waypoint_2" "breakAfter"
  movej(get_inverse_kin(Waypoint_2_p, qnear=Waypoint_2_q), a=1.3962634015954636, v=1.0471975511965976)
  $ 143 "MoveJ"
  $ 144 "Waypoint_13" "breakAfter"
  movej(get_inverse_kin(Waypoint_13_p, qnear=Waypoint_13_q), a=1.3962634015954636, v=1.0471975511965976)
  # begin: URCap Program Node
  #   Source: Robotiq_Grippers, 1.8.11.21258, Robotiq Inc.
  #   Type: Gripper
  $ 145 "Gripper Close (2)"
  if not(gripper_connected[1]):
    popup("Gripper 2 must be connected to run this program.", "No connection", False, True, True)
  end
  if not(rq_is_gripper_activated("2")):
    popup("Gripper 2 is not activated. Go to Installation tab > Gripper to activate it and run the program again.", "Not activated", False, True, True)
  end
  rq_set_pos_spd_for(255, 0, 0, "2")
  rq_wait_pos_spe_for_request(255, 0, 0, "2")
  rq_go_to("2")
  rq_wait("2")
  # end: URCap Program Node
  $ 146 "MoveJ"
  $ 147 "Waypoint_12" "breakAfter"
  movej(get_inverse_kin(Waypoint_12_p, qnear=Waypoint_12_q), a=1.3962634015954636, v=1.0471975511965976)
  # begin: URCap Program Node
  #   Source: Robotiq_Grippers, 1.8.11.21258, Robotiq Inc.
  #   Type: Gripper
  $ 148 "Gripper Open (2)"
  if not(gripper_connected[1]):
    popup("Gripper 2 must be connected to run this program.", "No connection", False, True, True)
  end
  if not(rq_is_gripper_activated("2")):
    popup("Gripper 2 is not activated. Go to Installation tab > Gripper to activate it and run the program again.", "Not activated", False, True, True)
  end
  rq_set_pos_spd_for(0, 0, 0, "2")
  rq_wait_pos_spe_for_request(0, 0, 0, "2")
  rq_go_to("2")
  rq_wait("2")
  # end: URCap Program Node
  $ 149 "Mouvement F"
  $ 150 "MoveJ"
  $ 151 "Waypoint_2" "breakAfter"
  movej(get_inverse_kin(Waypoint_2_p, qnear=Waypoint_2_q), a=1.3962634015954636, v=1.0471975511965976)
  $ 152 "MoveJ"
  $ 153 "Waypoint_14" "breakAfter"
  movej(get_inverse_kin(Waypoint_14_p, qnear=Waypoint_14_q), a=1.3962634015954636, v=1.0471975511965976)
  # begin: URCap Program Node
  #   Source: Robotiq_Grippers, 1.8.11.21258, Robotiq Inc.
  #   Type: Gripper
  $ 154 "Gripper Close (2)"
  if not(gripper_connected[1]):
    popup("Gripper 2 must be connected to run this program.", "No connection", False, True, True)
  end
  if not(rq_is_gripper_activated("2")):
    popup("Gripper 2 is not activated. Go to Installation tab > Gripper to activate it and run the program again.", "Not activated", False, True, True)
  end
  rq_set_pos_spd_for(255, 0, 0, "2")
  rq_wait_pos_spe_for_request(255, 0, 0, "2")
  rq_go_to("2")
  rq_wait("2")
  # end: URCap Program Node
  $ 155 "MoveJ"
  $ 156 "Waypoint_15" "breakAfter"
  movej(get_inverse_kin(Waypoint_15_p, qnear=Waypoint_15_q), a=1.3962634015954636, v=1.0471975511965976)
  $ 157 "MoveJ"
  $ 158 "Waypoint_23" "breakAfter"
  movej(get_inverse_kin(Waypoint_23_p, qnear=Waypoint_23_q), a=1.3962634015954636, v=1.0471975511965976)
  $ 159 "MoveJ"
  $ 160 "Waypoint_16" "breakAfter"
  movej(get_inverse_kin(Waypoint_16_p, qnear=Waypoint_16_q), a=1.3962634015954636, v=1.0471975511965976)
  # begin: URCap Program Node
  #   Source: Robotiq_Grippers, 1.8.11.21258, Robotiq Inc.
  #   Type: Gripper
  $ 161 "Gripper Open (2)"
  if not(gripper_connected[1]):
    popup("Gripper 2 must be connected to run this program.", "No connection", False, True, True)
  end
  if not(rq_is_gripper_activated("2")):
    popup("Gripper 2 is not activated. Go to Installation tab > Gripper to activate it and run the program again.", "Not activated", False, True, True)
  end
  rq_set_pos_spd_for(0, 0, 0, "2")
  rq_wait_pos_spe_for_request(0, 0, 0, "2")
  rq_go_to("2")
  rq_wait("2")
  # end: URCap Program Node
  $ 162 "MoveJ"
  $ 163 "Waypoint_2" "breakAfter"
  movej(get_inverse_kin(Waypoint_2_p, qnear=Waypoint_2_q), a=1.3962634015954636, v=1.0471975511965976)
  $ 164 "MoveJ"
  $ 165 "Waypoint_17" "breakAfter"
  movej(get_inverse_kin(Waypoint_17_p, qnear=Waypoint_17_q), a=1.3962634015954636, v=1.0471975511965976)
  # begin: URCap Program Node
  #   Source: Robotiq_Grippers, 1.8.11.21258, Robotiq Inc.
  #   Type: Gripper
  $ 166 "Gripper Close (2)"
  if not(gripper_connected[1]):
    popup("Gripper 2 must be connected to run this program.", "No connection", False, True, True)
  end
  if not(rq_is_gripper_activated("2")):
    popup("Gripper 2 is not activated. Go to Installation tab > Gripper to activate it and run the program again.", "Not activated", False, True, True)
  end
  rq_set_pos_spd_for(255, 0, 0, "2")
  rq_wait_pos_spe_for_request(255, 0, 0, "2")
  rq_go_to("2")
  rq_wait("2")
  # end: URCap Program Node
  $ 167 "MoveJ"
  $ 168 "Waypoint_18" "breakAfter"
  movej(get_inverse_kin(Waypoint_18_p, qnear=Waypoint_18_q), a=1.3962634015954636, v=1.0471975511965976)
  $ 169 "MoveJ"
  $ 170 "Waypoint_19" "breakAfter"
  movej(get_inverse_kin(Waypoint_19_p, qnear=Waypoint_19_q), a=1.3962634015954636, v=1.0471975511965976)
  $ 171 "MoveJ"
  $ 172 "Waypoint_20" "breakAfter"
  movej(get_inverse_kin(Waypoint_20_p, qnear=Waypoint_20_q), a=1.3962634015954636, v=1.0471975511965976)
  # begin: URCap Program Node
  #   Source: Robotiq_Grippers, 1.8.11.21258, Robotiq Inc.
  #   Type: Gripper
  $ 173 "Gripper Open (2)"
  if not(gripper_connected[1]):
    popup("Gripper 2 must be connected to run this program.", "No connection", False, True, True)
  end
  if not(rq_is_gripper_activated("2")):
    popup("Gripper 2 is not activated. Go to Installation tab > Gripper to activate it and run the program again.", "Not activated", False, True, True)
  end
  rq_set_pos_spd_for(0, 0, 0, "2")
  rq_wait_pos_spe_for_request(0, 0, 0, "2")
  rq_go_to("2")
  rq_wait("2")
  # end: URCap Program Node
  $ 174 "MoveJ"
  $ 175 "Waypoint_2" "breakAfter"
  movej(get_inverse_kin(Waypoint_2_p, qnear=Waypoint_2_q), a=1.3962634015954636, v=1.0471975511965976)
  $ 176 "MoveJ"
  $ 177 "Waypoint_21" "breakAfter"
  movej(get_inverse_kin(Waypoint_21_p, qnear=Waypoint_21_q), a=1.3962634015954636, v=1.0471975511965976)
  # begin: URCap Program Node
  #   Source: Robotiq_Grippers, 1.8.11.21258, Robotiq Inc.
  #   Type: Gripper
  $ 178 "Gripper Close (2)"
  if not(gripper_connected[1]):
    popup("Gripper 2 must be connected to run this program.", "No connection", False, True, True)
  end
  if not(rq_is_gripper_activated("2")):
    popup("Gripper 2 is not activated. Go to Installation tab > Gripper to activate it and run the program again.", "Not activated", False, True, True)
  end
  rq_set_pos_spd_for(255, 0, 0, "2")
  rq_wait_pos_spe_for_request(255, 0, 0, "2")
  rq_go_to("2")
  rq_wait("2")
  # end: URCap Program Node
  $ 179 "MoveJ"
  $ 180 "Waypoint_32" "breakAfter"
  movej(get_inverse_kin(Waypoint_32_p, qnear=Waypoint_32_q), a=1.3962634015954636, v=1.0471975511965976)
  $ 181 "MoveJ"
  $ 182 "MoveJ"
  $ 183 "Waypoint_2" "breakAfter"
  movej(get_inverse_kin(Waypoint_2_p, qnear=Waypoint_2_q), a=1.3962634015954636, v=1.0471975511965976)
  $ 184 "MoveJ"
  $ 185 "Waypoint_24" "breakAfter"
  movej(get_inverse_kin(Waypoint_24_p, qnear=Waypoint_24_q), a=1.3962634015954636, v=1.0471975511965976)
  # begin: URCap Program Node
  #   Source: Robotiq_Grippers, 1.8.11.21258, Robotiq Inc.
  #   Type: Gripper
  $ 186 "Gripper Close (2)"
  if not(gripper_connected[1]):
    popup("Gripper 2 must be connected to run this program.", "No connection", False, True, True)
  end
  if not(rq_is_gripper_activated("2")):
    popup("Gripper 2 is not activated. Go to Installation tab > Gripper to activate it and run the program again.", "Not activated", False, True, True)
  end
  rq_set_pos_spd_for(255, 0, 0, "2")
  rq_wait_pos_spe_for_request(255, 0, 0, "2")
  rq_go_to("2")
  rq_wait("2")
  # end: URCap Program Node
  $ 187 "MoveJ"
  $ 188 "Waypoint_25" "breakAfter"
  movej(get_inverse_kin(Waypoint_25_p, qnear=Waypoint_25_q), a=1.3962634015954636, v=1.0471975511965976)
  $ 189 "MoveJ"
  $ 190 "Waypoint_27" "breakAfter"
  movej(get_inverse_kin(Waypoint_27_p, qnear=Waypoint_27_q), a=1.3962634015954636, v=1.0471975511965976)
  $ 191 "MoveJ"
  $ 192 "Waypoint_26" "breakAfter"
  movej(get_inverse_kin(Waypoint_26_p, qnear=Waypoint_26_q), a=1.3962634015954636, v=1.0471975511965976)
  # begin: URCap Program Node
  #   Source: Robotiq_Grippers, 1.8.11.21258, Robotiq Inc.
  #   Type: Gripper
  $ 193 "Gripper Open (2)"
  if not(gripper_connected[1]):
    popup("Gripper 2 must be connected to run this program.", "No connection", False, True, True)
  end
  if not(rq_is_gripper_activated("2")):
    popup("Gripper 2 is not activated. Go to Installation tab > Gripper to activate it and run the program again.", "Not activated", False, True, True)
  end
  rq_set_pos_spd_for(0, 0, 0, "2")
  rq_wait_pos_spe_for_request(0, 0, 0, "2")
  rq_go_to("2")
  rq_wait("2")
  # end: URCap Program Node
  $ 194 "MoveJ"
  $ 195 "Waypoint_2" "breakAfter"
  movej(get_inverse_kin(Waypoint_2_p, qnear=Waypoint_2_q), a=1.3962634015954636, v=1.0471975511965976)
  $ 196 "MoveJ"
  $ 197 "Waypoint_28" "breakAfter"
  movej(get_inverse_kin(Waypoint_28_p, qnear=Waypoint_28_q), a=1.3962634015954636, v=1.0471975511965976)
  # begin: URCap Program Node
  #   Source: Robotiq_Grippers, 1.8.11.21258, Robotiq Inc.
  #   Type: Gripper
  $ 198 "Gripper Close (2)"
  if not(gripper_connected[1]):
    popup("Gripper 2 must be connected to run this program.", "No connection", False, True, True)
  end
  if not(rq_is_gripper_activated("2")):
    popup("Gripper 2 is not activated. Go to Installation tab > Gripper to activate it and run the program again.", "Not activated", False, True, True)
  end
  rq_set_pos_spd_for(255, 0, 0, "2")
  rq_wait_pos_spe_for_request(255, 0, 0, "2")
  rq_go_to("2")
  rq_wait("2")
  # end: URCap Program Node
  $ 199 "MoveJ"
  $ 200 "Waypoint_29" "breakAfter"
  movej(get_inverse_kin(Waypoint_29_p, qnear=Waypoint_29_q), a=1.3962634015954636, v=1.0471975511965976)
  $ 201 "MoveJ"
  $ 202 "Waypoint_30" "breakAfter"
  movej(get_inverse_kin(Waypoint_30_p, qnear=Waypoint_30_q), a=1.3962634015954636, v=1.0471975511965976)
  $ 203 "MoveJ"
  $ 204 "Waypoint_31" "breakAfter"
  movej(get_inverse_kin(Waypoint_31_p, qnear=Waypoint_31_q), a=1.3962634015954636, v=1.0471975511965976)
  # begin: URCap Program Node
  #   Source: Robotiq_Grippers, 1.8.11.21258, Robotiq Inc.
  #   Type: Gripper
  $ 205 "Gripper Open (2)"
  if not(gripper_connected[1]):
    popup("Gripper 2 must be connected to run this program.", "No connection", False, True, True)
  end
  if not(rq_is_gripper_activated("2")):
    popup("Gripper 2 is not activated. Go to Installation tab > Gripper to activate it and run the program again.", "Not activated", False, True, True)
  end
  rq_set_pos_spd_for(0, 0, 0, "2")
  rq_wait_pos_spe_for_request(0, 0, 0, "2")
  rq_go_to("2")
  rq_wait("2")
  # end: URCap Program Node
  $ 206 "MoveJ"
  $ 207 "Waypoint_2" "breakAfter"
  movej(get_inverse_kin(Waypoint_2_p, qnear=Waypoint_2_q), a=1.3962634015954636, v=1.0471975511965976)
  $ 208 "Mouvement F'"
  $ 209 "MoveJ"
  $ 210 "Waypoint_2" "breakAfter"
  movej(get_inverse_kin(Waypoint_2_p, qnear=Waypoint_2_q), a=1.3962634015954636, v=1.0471975511965976)
  $ 211 "MoveJ"
  $ 212 "Waypoint_14" "breakAfter"
  movej(get_inverse_kin(Waypoint_14_p, qnear=Waypoint_14_q), a=1.3962634015954636, v=1.0471975511965976)
  # begin: URCap Program Node
  #   Source: Robotiq_Grippers, 1.8.11.21258, Robotiq Inc.
  #   Type: Gripper
  $ 213 "Gripper Close (2)"
  if not(gripper_connected[1]):
    popup("Gripper 2 must be connected to run this program.", "No connection", False, True, True)
  end
  if not(rq_is_gripper_activated("2")):
    popup("Gripper 2 is not activated. Go to Installation tab > Gripper to activate it and run the program again.", "Not activated", False, True, True)
  end
  rq_set_pos_spd_for(255, 0, 0, "2")
  rq_wait_pos_spe_for_request(255, 0, 0, "2")
  rq_go_to("2")
  rq_wait("2")
  # end: URCap Program Node
  $ 214 "MoveJ"
  $ 215 "Waypoint_15" "breakAfter"
  movej(get_inverse_kin(Waypoint_15_p, qnear=Waypoint_15_q), a=1.3962634015954636, v=1.0471975511965976)
  $ 216 "MoveJ"
  $ 217 "Waypoint_23" "breakAfter"
  movej(get_inverse_kin(Waypoint_23_p, qnear=Waypoint_23_q), a=1.3962634015954636, v=1.0471975511965976)
  $ 218 "MoveJ"
  $ 219 "Waypoint_16" "breakAfter"
  movej(get_inverse_kin(Waypoint_16_p, qnear=Waypoint_16_q), a=1.3962634015954636, v=1.0471975511965976)
  # begin: URCap Program Node
  #   Source: Robotiq_Grippers, 1.8.11.21258, Robotiq Inc.
  #   Type: Gripper
  $ 220 "Gripper Open (2)"
  if not(gripper_connected[1]):
    popup("Gripper 2 must be connected to run this program.", "No connection", False, True, True)
  end
  if not(rq_is_gripper_activated("2")):
    popup("Gripper 2 is not activated. Go to Installation tab > Gripper to activate it and run the program again.", "Not activated", False, True, True)
  end
  rq_set_pos_spd_for(0, 0, 0, "2")
  rq_wait_pos_spe_for_request(0, 0, 0, "2")
  rq_go_to("2")
  rq_wait("2")
  # end: URCap Program Node
  $ 221 "MoveJ"
  $ 222 "Waypoint_2" "breakAfter"
  movej(get_inverse_kin(Waypoint_2_p, qnear=Waypoint_2_q), a=1.3962634015954636, v=1.0471975511965976)
  $ 223 "MoveJ"
  $ 224 "Waypoint_17" "breakAfter"
  movej(get_inverse_kin(Waypoint_17_p, qnear=Waypoint_17_q), a=1.3962634015954636, v=1.0471975511965976)
  # begin: URCap Program Node
  #   Source: Robotiq_Grippers, 1.8.11.21258, Robotiq Inc.
  #   Type: Gripper
  $ 225 "Gripper Close (2)"
  if not(gripper_connected[1]):
    popup("Gripper 2 must be connected to run this program.", "No connection", False, True, True)
  end
  if not(rq_is_gripper_activated("2")):
    popup("Gripper 2 is not activated. Go to Installation tab > Gripper to activate it and run the program again.", "Not activated", False, True, True)
  end
  rq_set_pos_spd_for(255, 0, 0, "2")
  rq_wait_pos_spe_for_request(255, 0, 0, "2")
  rq_go_to("2")
  rq_wait("2")
  # end: URCap Program Node
  $ 226 "MoveJ"
  $ 227 "Waypoint_18" "breakAfter"
  movej(get_inverse_kin(Waypoint_18_p, qnear=Waypoint_18_q), a=1.3962634015954636, v=1.0471975511965976)
  $ 228 "MoveJ"
  $ 229 "Waypoint_19" "breakAfter"
  movej(get_inverse_kin(Waypoint_19_p, qnear=Waypoint_19_q), a=1.3962634015954636, v=1.0471975511965976)
  $ 230 "MoveJ"
  $ 231 "Waypoint_20" "breakAfter"
  movej(get_inverse_kin(Waypoint_20_p, qnear=Waypoint_20_q), a=1.3962634015954636, v=1.0471975511965976)
  # begin: URCap Program Node
  #   Source: Robotiq_Grippers, 1.8.11.21258, Robotiq Inc.
  #   Type: Gripper
  $ 232 "Gripper Open (2)"
  if not(gripper_connected[1]):
    popup("Gripper 2 must be connected to run this program.", "No connection", False, True, True)
  end
  if not(rq_is_gripper_activated("2")):
    popup("Gripper 2 is not activated. Go to Installation tab > Gripper to activate it and run the program again.", "Not activated", False, True, True)
  end
  rq_set_pos_spd_for(0, 0, 0, "2")
  rq_wait_pos_spe_for_request(0, 0, 0, "2")
  rq_go_to("2")
  rq_wait("2")
  # end: URCap Program Node
  $ 233 "MoveJ"
  $ 234 "Waypoint_2" "breakAfter"
  movej(get_inverse_kin(Waypoint_2_p, qnear=Waypoint_2_q), a=1.3962634015954636, v=1.0471975511965976)
  $ 235 "MoveJ"
  $ 236 "Waypoint_21" "breakAfter"
  movej(get_inverse_kin(Waypoint_21_p, qnear=Waypoint_21_q), a=1.3962634015954636, v=1.0471975511965976)
  # begin: URCap Program Node
  #   Source: Robotiq_Grippers, 1.8.11.21258, Robotiq Inc.
  #   Type: Gripper
  $ 237 "Gripper Close (2)"
  if not(gripper_connected[1]):
    popup("Gripper 2 must be connected to run this program.", "No connection", False, True, True)
  end
  if not(rq_is_gripper_activated("2")):
    popup("Gripper 2 is not activated. Go to Installation tab > Gripper to activate it and run the program again.", "Not activated", False, True, True)
  end
  rq_set_pos_spd_for(255, 0, 0, "2")
  rq_wait_pos_spe_for_request(255, 0, 0, "2")
  rq_go_to("2")
  rq_wait("2")
  # end: URCap Program Node
  $ 238 "MoveJ"
  $ 239 "Waypoint_22" "breakAfter"
  movej(get_inverse_kin(Waypoint_22_p, qnear=Waypoint_22_q), a=1.3962634015954636, v=1.0471975511965976)
  # begin: URCap Program Node
  #   Source: Robotiq_Grippers, 1.8.11.21258, Robotiq Inc.
  #   Type: Gripper
  $ 240 "Gripper Open (2)"
  if not(gripper_connected[1]):
    popup("Gripper 2 must be connected to run this program.", "No connection", False, True, True)
  end
  if not(rq_is_gripper_activated("2")):
    popup("Gripper 2 is not activated. Go to Installation tab > Gripper to activate it and run the program again.", "Not activated", False, True, True)
  end
  rq_set_pos_spd_for(0, 0, 0, "2")
  rq_wait_pos_spe_for_request(0, 0, 0, "2")
  rq_go_to("2")
  rq_wait("2")
  # end: URCap Program Node
  $ 241 "MoveJ"
  $ 242 "MoveJ"
  $ 243 "Waypoint_2" "breakAfter"
  movej(get_inverse_kin(Waypoint_2_p, qnear=Waypoint_2_q), a=1.3962634015954636, v=1.0471975511965976)
  $ 244 "MoveJ"
  $ 245 "Waypoint_24" "breakAfter"
  movej(get_inverse_kin(Waypoint_24_p, qnear=Waypoint_24_q), a=1.3962634015954636, v=1.0471975511965976)
  # begin: URCap Program Node
  #   Source: Robotiq_Grippers, 1.8.11.21258, Robotiq Inc.
  #   Type: Gripper
  $ 246 "Gripper Close (2)"
  if not(gripper_connected[1]):
    popup("Gripper 2 must be connected to run this program.", "No connection", False, True, True)
  end
  if not(rq_is_gripper_activated("2")):
    popup("Gripper 2 is not activated. Go to Installation tab > Gripper to activate it and run the program again.", "Not activated", False, True, True)
  end
  rq_set_pos_spd_for(255, 0, 0, "2")
  rq_wait_pos_spe_for_request(255, 0, 0, "2")
  rq_go_to("2")
  rq_wait("2")
  # end: URCap Program Node
  $ 247 "MoveJ"
  $ 248 "Waypoint_25" "breakAfter"
  movej(get_inverse_kin(Waypoint_25_p, qnear=Waypoint_25_q), a=1.3962634015954636, v=1.0471975511965976)
  $ 249 "MoveJ"
  $ 250 "Waypoint_27" "breakAfter"
  movej(get_inverse_kin(Waypoint_27_p, qnear=Waypoint_27_q), a=1.3962634015954636, v=1.0471975511965976)
  $ 251 "MoveJ"
  $ 252 "Waypoint_26" "breakAfter"
  movej(get_inverse_kin(Waypoint_26_p, qnear=Waypoint_26_q), a=1.3962634015954636, v=1.0471975511965976)
  # begin: URCap Program Node
  #   Source: Robotiq_Grippers, 1.8.11.21258, Robotiq Inc.
  #   Type: Gripper
  $ 253 "Gripper Open (2)"
  if not(gripper_connected[1]):
    popup("Gripper 2 must be connected to run this program.", "No connection", False, True, True)
  end
  if not(rq_is_gripper_activated("2")):
    popup("Gripper 2 is not activated. Go to Installation tab > Gripper to activate it and run the program again.", "Not activated", False, True, True)
  end
  rq_set_pos_spd_for(0, 0, 0, "2")
  rq_wait_pos_spe_for_request(0, 0, 0, "2")
  rq_go_to("2")
  rq_wait("2")
  # end: URCap Program Node
  $ 254 "MoveJ"
  $ 255 "Waypoint_2" "breakAfter"
  movej(get_inverse_kin(Waypoint_2_p, qnear=Waypoint_2_q), a=1.3962634015954636, v=1.0471975511965976)
  $ 256 "MoveJ"
  $ 257 "Waypoint_28" "breakAfter"
  movej(get_inverse_kin(Waypoint_28_p, qnear=Waypoint_28_q), a=1.3962634015954636, v=1.0471975511965976)
  # begin: URCap Program Node
  #   Source: Robotiq_Grippers, 1.8.11.21258, Robotiq Inc.
  #   Type: Gripper
  $ 258 "Gripper Close (2)"
  if not(gripper_connected[1]):
    popup("Gripper 2 must be connected to run this program.", "No connection", False, True, True)
  end
  if not(rq_is_gripper_activated("2")):
    popup("Gripper 2 is not activated. Go to Installation tab > Gripper to activate it and run the program again.", "Not activated", False, True, True)
  end
  rq_set_pos_spd_for(255, 0, 0, "2")
  rq_wait_pos_spe_for_request(255, 0, 0, "2")
  rq_go_to("2")
  rq_wait("2")
  # end: URCap Program Node
  $ 259 "MoveJ"
  $ 260 "Waypoint_29" "breakAfter"
  movej(get_inverse_kin(Waypoint_29_p, qnear=Waypoint_29_q), a=1.3962634015954636, v=1.0471975511965976)
  $ 261 "MoveJ"
  $ 262 "Waypoint_30" "breakAfter"
  movej(get_inverse_kin(Waypoint_30_p, qnear=Waypoint_30_q), a=1.3962634015954636, v=1.0471975511965976)
  $ 263 "MoveJ"
  $ 264 "Waypoint_31" "breakAfter"
  movej(get_inverse_kin(Waypoint_31_p, qnear=Waypoint_31_q), a=1.3962634015954636, v=1.0471975511965976)
  # begin: URCap Program Node
  #   Source: Robotiq_Grippers, 1.8.11.21258, Robotiq Inc.
  #   Type: Gripper
  $ 265 "Gripper Open (2)"
  if not(gripper_connected[1]):
    popup("Gripper 2 must be connected to run this program.", "No connection", False, True, True)
  end
  if not(rq_is_gripper_activated("2")):
    popup("Gripper 2 is not activated. Go to Installation tab > Gripper to activate it and run the program again.", "Not activated", False, True, True)
  end
  rq_set_pos_spd_for(0, 0, 0, "2")
  rq_wait_pos_spe_for_request(0, 0, 0, "2")
  rq_go_to("2")
  rq_wait("2")
  # end: URCap Program Node
  $ 266 "MoveJ"
  $ 267 "Waypoint_2" "breakAfter"
  movej(get_inverse_kin(Waypoint_2_p, qnear=Waypoint_2_q), a=1.3962634015954636, v=1.0471975511965976)
  $ 268 "Mouvement B'"
  $ 269 "MoveJ"
  $ 270 "Waypoint_2" "breakAfter"
  movej(get_inverse_kin(Waypoint_2_p, qnear=Waypoint_2_q), a=1.3962634015954636, v=1.0471975511965976)
  $ 271 "MoveJ"
  $ 272 "Waypoint_14" "breakAfter"
  movej(get_inverse_kin(Waypoint_14_p, qnear=Waypoint_14_q), a=1.3962634015954636, v=1.0471975511965976)
  # begin: URCap Program Node
  #   Source: Robotiq_Grippers, 1.8.11.21258, Robotiq Inc.
  #   Type: Gripper
  $ 273 "Gripper Close (2)"
  if not(gripper_connected[1]):
    popup("Gripper 2 must be connected to run this program.", "No connection", False, True, True)
  end
  if not(rq_is_gripper_activated("2")):
    popup("Gripper 2 is not activated. Go to Installation tab > Gripper to activate it and run the program again.", "Not activated", False, True, True)
  end
  rq_set_pos_spd_for(255, 0, 0, "2")
  rq_wait_pos_spe_for_request(255, 0, 0, "2")
  rq_go_to("2")
  rq_wait("2")
  # end: URCap Program Node
  $ 274 "MoveJ"
  $ 275 "Waypoint_15" "breakAfter"
  movej(get_inverse_kin(Waypoint_15_p, qnear=Waypoint_15_q), a=1.3962634015954636, v=1.0471975511965976)
  $ 276 "MoveJ"
  $ 277 "Waypoint_33" "breakAfter"
  movej(get_inverse_kin(Waypoint_33_p, qnear=Waypoint_33_q), a=1.3962634015954636, v=1.0471975511965976)
  $ 278 "MoveJ"
  $ 279 "Waypoint_34" "breakAfter"
  movej(get_inverse_kin(Waypoint_34_p, qnear=Waypoint_34_q), a=1.3962634015954636, v=1.0471975511965976)
  # begin: URCap Program Node
  #   Source: Robotiq_Grippers, 1.8.11.21258, Robotiq Inc.
  #   Type: Gripper
  $ 280 "Gripper Open (2)"
  if not(gripper_connected[1]):
    popup("Gripper 2 must be connected to run this program.", "No connection", False, True, True)
  end
  if not(rq_is_gripper_activated("2")):
    popup("Gripper 2 is not activated. Go to Installation tab > Gripper to activate it and run the program again.", "Not activated", False, True, True)
  end
  rq_set_pos_spd_for(0, 0, 0, "2")
  rq_wait_pos_spe_for_request(0, 0, 0, "2")
  rq_go_to("2")
  rq_wait("2")
  # end: URCap Program Node
  $ 281 "MoveJ"
  $ 282 "Waypoint_2" "breakAfter"
  movej(get_inverse_kin(Waypoint_2_p, qnear=Waypoint_2_q), a=1.3962634015954636, v=1.0471975511965976)
  $ 283 "MoveJ"
  $ 284 "Waypoint_14" "breakAfter"
  movej(get_inverse_kin(Waypoint_14_p, qnear=Waypoint_14_q), a=1.3962634015954636, v=1.0471975511965976)
  # begin: URCap Program Node
  #   Source: Robotiq_Grippers, 1.8.11.21258, Robotiq Inc.
  #   Type: Gripper
  $ 285 "Gripper Close (2)"
  if not(gripper_connected[1]):
    popup("Gripper 2 must be connected to run this program.", "No connection", False, True, True)
  end
  if not(rq_is_gripper_activated("2")):
    popup("Gripper 2 is not activated. Go to Installation tab > Gripper to activate it and run the program again.", "Not activated", False, True, True)
  end
  rq_set_pos_spd_for(255, 0, 0, "2")
  rq_wait_pos_spe_for_request(255, 0, 0, "2")
  rq_go_to("2")
  rq_wait("2")
  # end: URCap Program Node
  $ 286 "MoveJ"
  $ 287 "Waypoint_15" "breakAfter"
  movej(get_inverse_kin(Waypoint_15_p, qnear=Waypoint_15_q), a=1.3962634015954636, v=1.0471975511965976)
  $ 288 "MoveJ"
  $ 289 "Waypoint_35" "breakAfter"
  movej(get_inverse_kin(Waypoint_35_p, qnear=Waypoint_35_q), a=1.3962634015954636, v=1.0471975511965976)
  $ 290 "MoveJ"
  $ 291 "Waypoint_36" "breakAfter"
  movej(get_inverse_kin(Waypoint_36_p, qnear=Waypoint_36_q), a=1.3962634015954636, v=1.0471975511965976)
  # begin: URCap Program Node
  #   Source: Robotiq_Grippers, 1.8.11.21258, Robotiq Inc.
  #   Type: Gripper
  $ 292 "Gripper Open (2)"
  if not(gripper_connected[1]):
    popup("Gripper 2 must be connected to run this program.", "No connection", False, True, True)
  end
  if not(rq_is_gripper_activated("2")):
    popup("Gripper 2 is not activated. Go to Installation tab > Gripper to activate it and run the program again.", "Not activated", False, True, True)
  end
  rq_set_pos_spd_for(0, 0, 0, "2")
  rq_wait_pos_spe_for_request(0, 0, 0, "2")
  rq_go_to("2")
  rq_wait("2")
  # end: URCap Program Node
  $ 293 "MoveJ"
  $ 294 "Waypoint_37" "breakAfter"
  movej(get_inverse_kin(Waypoint_37_p, qnear=Waypoint_37_q), a=1.3962634015954636, v=1.0471975511965976)
  # begin: URCap Program Node
  #   Source: Robotiq_Grippers, 1.8.11.21258, Robotiq Inc.
  #   Type: Gripper
  $ 295 "Gripper Close (2)"
  if not(gripper_connected[1]):
    popup("Gripper 2 must be connected to run this program.", "No connection", False, True, True)
  end
  if not(rq_is_gripper_activated("2")):
    popup("Gripper 2 is not activated. Go to Installation tab > Gripper to activate it and run the program again.", "Not activated", False, True, True)
  end
  rq_set_pos_spd_for(255, 0, 0, "2")
  rq_wait_pos_spe_for_request(255, 0, 0, "2")
  rq_go_to("2")
  rq_wait("2")
  # end: URCap Program Node
  $ 296 "MoveJ"
  $ 297 "Waypoint_38" "breakAfter"
  movej(get_inverse_kin(Waypoint_38_p, qnear=Waypoint_38_q), a=1.3962634015954636, v=1.0471975511965976)
  # begin: URCap Program Node
  #   Source: Robotiq_Grippers, 1.8.11.21258, Robotiq Inc.
  #   Type: Gripper
  $ 298 "Gripper Open (2)"
  if not(gripper_connected[1]):
    popup("Gripper 2 must be connected to run this program.", "No connection", False, True, True)
  end
  if not(rq_is_gripper_activated("2")):
    popup("Gripper 2 is not activated. Go to Installation tab > Gripper to activate it and run the program again.", "Not activated", False, True, True)
  end
  rq_set_pos_spd_for(0, 0, 0, "2")
  rq_wait_pos_spe_for_request(0, 0, 0, "2")
  rq_go_to("2")
  rq_wait("2")
  # end: URCap Program Node
  $ 299 "MoveJ"
  $ 300 "Waypoint_39" "breakAfter"
  movej(get_inverse_kin(Waypoint_39_p, qnear=Waypoint_39_q), a=1.3962634015954636, v=1.0471975511965976)
  # begin: URCap Program Node
  #   Source: Robotiq_Grippers, 1.8.11.21258, Robotiq Inc.
  #   Type: Gripper
  $ 301 "Gripper Close (2)"
  if not(gripper_connected[1]):
    popup("Gripper 2 must be connected to run this program.", "No connection", False, True, True)
  end
  if not(rq_is_gripper_activated("2")):
    popup("Gripper 2 is not activated. Go to Installation tab > Gripper to activate it and run the program again.", "Not activated", False, True, True)
  end
  rq_set_pos_spd_for(255, 0, 0, "2")
  rq_wait_pos_spe_for_request(255, 0, 0, "2")
  rq_go_to("2")
  rq_wait("2")
  # end: URCap Program Node
  $ 302 "MoveJ"
  $ 303 "Waypoint_40" "breakAfter"
  movej(get_inverse_kin(Waypoint_40_p, qnear=Waypoint_40_q), a=1.3962634015954636, v=1.0471975511965976)
  $ 304 "MoveJ"
  $ 305 "Waypoint_41" "breakAfter"
  movej(get_inverse_kin(Waypoint_41_p, qnear=Waypoint_41_q), a=1.3962634015954636, v=1.0471975511965976)
  $ 306 "MoveJ"
  $ 307 "Waypoint_42" "breakAfter"
  movej(get_inverse_kin(Waypoint_42_p, qnear=Waypoint_42_q), a=1.3962634015954636, v=1.0471975511965976)
  # begin: URCap Program Node
  #   Source: Robotiq_Grippers, 1.8.11.21258, Robotiq Inc.
  #   Type: Gripper
  $ 308 "Gripper Open (2)"
  if not(gripper_connected[1]):
    popup("Gripper 2 must be connected to run this program.", "No connection", False, True, True)
  end
  if not(rq_is_gripper_activated("2")):
    popup("Gripper 2 is not activated. Go to Installation tab > Gripper to activate it and run the program again.", "Not activated", False, True, True)
  end
  rq_set_pos_spd_for(0, 0, 0, "2")
  rq_wait_pos_spe_for_request(0, 0, 0, "2")
  rq_go_to("2")
  rq_wait("2")
  # end: URCap Program Node
  $ 309 "MoveJ"
  $ 310 "Waypoint_2" "breakAfter"
  movej(get_inverse_kin(Waypoint_2_p, qnear=Waypoint_2_q), a=1.3962634015954636, v=1.0471975511965976)
  $ 311 "MoveJ"
  $ 312 "Waypoint_14" "breakAfter"
  movej(get_inverse_kin(Waypoint_14_p, qnear=Waypoint_14_q), a=1.3962634015954636, v=1.0471975511965976)
  # begin: URCap Program Node
  #   Source: Robotiq_Grippers, 1.8.11.21258, Robotiq Inc.
  #   Type: Gripper
  $ 313 "Gripper Close (2)"
  if not(gripper_connected[1]):
    popup("Gripper 2 must be connected to run this program.", "No connection", False, True, True)
  end
  if not(rq_is_gripper_activated("2")):
    popup("Gripper 2 is not activated. Go to Installation tab > Gripper to activate it and run the program again.", "Not activated", False, True, True)
  end
  rq_set_pos_spd_for(255, 0, 0, "2")
  rq_wait_pos_spe_for_request(255, 0, 0, "2")
  rq_go_to("2")
  rq_wait("2")
  # end: URCap Program Node
  $ 314 "MoveJ"
  $ 315 "Waypoint_43" "breakAfter"
  movej(get_inverse_kin(Waypoint_43_p, qnear=Waypoint_43_q), a=1.3962634015954636, v=1.0471975511965976)
  $ 316 "MoveJ"
  $ 317 "Waypoint_44" "breakAfter"
  movej(get_inverse_kin(Waypoint_44_p, qnear=Waypoint_44_q), a=1.3962634015954636, v=1.0471975511965976)
  $ 318 "MoveJ"
  $ 319 "Waypoint_45" "breakAfter"
  movej(get_inverse_kin(Waypoint_45_p, qnear=Waypoint_45_q), a=1.3962634015954636, v=1.0471975511965976)
  # begin: URCap Program Node
  #   Source: Robotiq_Grippers, 1.8.11.21258, Robotiq Inc.
  #   Type: Gripper
  $ 320 "Gripper Open (2)"
  if not(gripper_connected[1]):
    popup("Gripper 2 must be connected to run this program.", "No connection", False, True, True)
  end
  if not(rq_is_gripper_activated("2")):
    popup("Gripper 2 is not activated. Go to Installation tab > Gripper to activate it and run the program again.", "Not activated", False, True, True)
  end
  rq_set_pos_spd_for(0, 0, 0, "2")
  rq_wait_pos_spe_for_request(0, 0, 0, "2")
  rq_go_to("2")
  rq_wait("2")
  # end: URCap Program Node
  $ 321 "MoveJ"
  $ 322 "Waypoint_2" "breakAfter"
  movej(get_inverse_kin(Waypoint_2_p, qnear=Waypoint_2_q), a=1.3962634015954636, v=1.0471975511965976)
  $ 323 "MoveJ"
  $ 324 "Waypoint_14" "breakAfter"
  movej(get_inverse_kin(Waypoint_14_p, qnear=Waypoint_14_q), a=1.3962634015954636, v=1.0471975511965976)
  # begin: URCap Program Node
  #   Source: Robotiq_Grippers, 1.8.11.21258, Robotiq Inc.
  #   Type: Gripper
  $ 325 "Gripper Close (2)"
  if not(gripper_connected[1]):
    popup("Gripper 2 must be connected to run this program.", "No connection", False, True, True)
  end
  if not(rq_is_gripper_activated("2")):
    popup("Gripper 2 is not activated. Go to Installation tab > Gripper to activate it and run the program again.", "Not activated", False, True, True)
  end
  rq_set_pos_spd_for(255, 0, 0, "2")
  rq_wait_pos_spe_for_request(255, 0, 0, "2")
  rq_go_to("2")
  rq_wait("2")
  # end: URCap Program Node
  $ 326 "MoveJ"
  $ 327 "Waypoint_46" "breakAfter"
  movej(get_inverse_kin(Waypoint_46_p, qnear=Waypoint_46_q), a=1.3962634015954636, v=1.0471975511965976)
  $ 328 "MoveJ"
  $ 329 "Waypoint_47" "breakAfter"
  movej(get_inverse_kin(Waypoint_47_p, qnear=Waypoint_47_q), a=1.3962634015954636, v=1.0471975511965976)
  $ 330 "MoveJ"
  $ 331 "Waypoint_48" "breakAfter"
  movej(get_inverse_kin(Waypoint_48_p, qnear=Waypoint_48_q), a=1.3962634015954636, v=1.0471975511965976)
  # begin: URCap Program Node
  #   Source: Robotiq_Grippers, 1.8.11.21258, Robotiq Inc.
  #   Type: Gripper
  $ 332 "Gripper Open (2)"
  if not(gripper_connected[1]):
    popup("Gripper 2 must be connected to run this program.", "No connection", False, True, True)
  end
  if not(rq_is_gripper_activated("2")):
    popup("Gripper 2 is not activated. Go to Installation tab > Gripper to activate it and run the program again.", "Not activated", False, True, True)
  end
  rq_set_pos_spd_for(0, 0, 0, "2")
  rq_wait_pos_spe_for_request(0, 0, 0, "2")
  rq_go_to("2")
  rq_wait("2")
  # end: URCap Program Node
  $ 333 "MoveJ"
  $ 334 "Waypoint_2" "breakAfter"
  movej(get_inverse_kin(Waypoint_2_p, qnear=Waypoint_2_q), a=1.3962634015954636, v=1.0471975511965976)
  $ 335 "MoveJ"
  $ 336 "Waypoint_52" "breakAfter"
  movej(get_inverse_kin(Waypoint_52_p, qnear=Waypoint_52_q), a=1.3962634015954636, v=1.0471975511965976)
  # begin: URCap Program Node
  #   Source: Robotiq_Grippers, 1.8.11.21258, Robotiq Inc.
  #   Type: Gripper
  $ 337 "Gripper Close (2)"
  if not(gripper_connected[1]):
    popup("Gripper 2 must be connected to run this program.", "No connection", False, True, True)
  end
  if not(rq_is_gripper_activated("2")):
    popup("Gripper 2 is not activated. Go to Installation tab > Gripper to activate it and run the program again.", "Not activated", False, True, True)
  end
  rq_set_pos_spd_for(255, 0, 0, "2")
  rq_wait_pos_spe_for_request(255, 0, 0, "2")
  rq_go_to("2")
  rq_wait("2")
  # end: URCap Program Node
  $ 338 "MoveJ"
  $ 339 "Waypoint_49" "breakAfter"
  movej(get_inverse_kin(Waypoint_49_p, qnear=Waypoint_49_q), a=1.3962634015954636, v=1.0471975511965976)
  $ 340 "MoveJ"
  $ 341 "Waypoint_50" "breakAfter"
  movej(get_inverse_kin(Waypoint_50_p, qnear=Waypoint_50_q), a=1.3962634015954636, v=1.0471975511965976)
  # begin: URCap Program Node
  #   Source: Robotiq_Grippers, 1.8.11.21258, Robotiq Inc.
  #   Type: Gripper
  $ 342 "Gripper Open (2)"
  if not(gripper_connected[1]):
    popup("Gripper 2 must be connected to run this program.", "No connection", False, True, True)
  end
  if not(rq_is_gripper_activated("2")):
    popup("Gripper 2 is not activated. Go to Installation tab > Gripper to activate it and run the program again.", "Not activated", False, True, True)
  end
  rq_set_pos_spd_for(0, 0, 0, "2")
  rq_wait_pos_spe_for_request(0, 0, 0, "2")
  rq_go_to("2")
  rq_wait("2")
  # end: URCap Program Node
  $ 343 "MoveJ"
  $ 344 "Waypoint_2" "breakAfter"
  movej(get_inverse_kin(Waypoint_2_p, qnear=Waypoint_2_q), a=1.3962634015954636, v=1.0471975511965976)
  $ 345 "MoveJ"
  $ 346 "Waypoint_14" "breakAfter"
  movej(get_inverse_kin(Waypoint_14_p, qnear=Waypoint_14_q), a=1.3962634015954636, v=1.0471975511965976)
  # begin: URCap Program Node
  #   Source: Robotiq_Grippers, 1.8.11.21258, Robotiq Inc.
  #   Type: Gripper
  $ 347 "Gripper Close (2)"
  if not(gripper_connected[1]):
    popup("Gripper 2 must be connected to run this program.", "No connection", False, True, True)
  end
  if not(rq_is_gripper_activated("2")):
    popup("Gripper 2 is not activated. Go to Installation tab > Gripper to activate it and run the program again.", "Not activated", False, True, True)
  end
  rq_set_pos_spd_for(255, 0, 0, "2")
  rq_wait_pos_spe_for_request(255, 0, 0, "2")
  rq_go_to("2")
  rq_wait("2")
  # end: URCap Program Node
  $ 348 "MoveJ"
  $ 349 "Waypoint_51" "breakAfter"
  movej(get_inverse_kin(Waypoint_51_p, qnear=Waypoint_51_q), a=1.3962634015954636, v=1.0471975511965976)
  $ 350 "MoveJ"
  $ 351 "Waypoint_53" "breakAfter"
  movej(get_inverse_kin(Waypoint_53_p, qnear=Waypoint_53_q), a=1.3962634015954636, v=1.0471975511965976)
  # begin: URCap Program Node
  #   Source: Robotiq_Grippers, 1.8.11.21258, Robotiq Inc.
  #   Type: Gripper
  $ 352 "Gripper Open (2)"
  if not(gripper_connected[1]):
    popup("Gripper 2 must be connected to run this program.", "No connection", False, True, True)
  end
  if not(rq_is_gripper_activated("2")):
    popup("Gripper 2 is not activated. Go to Installation tab > Gripper to activate it and run the program again.", "Not activated", False, True, True)
  end
  rq_set_pos_spd_for(0, 0, 0, "2")
  rq_wait_pos_spe_for_request(0, 0, 0, "2")
  rq_go_to("2")
  rq_wait("2")
  # end: URCap Program Node
  $ 353 "MoveJ"
  $ 354 "Waypoint_2" "breakAfter"
  movej(get_inverse_kin(Waypoint_2_p, qnear=Waypoint_2_q), a=1.3962634015954636, v=1.0471975511965976)
  $ 355 "Mouvement B"
  $ 356 "MoveJ"
  $ 357 "Waypoint_2" "breakAfter"
  movej(get_inverse_kin(Waypoint_2_p, qnear=Waypoint_2_q), a=1.3962634015954636, v=1.0471975511965976)
  $ 358 "MoveJ"
  $ 359 "Waypoint_14" "breakAfter"
  movej(get_inverse_kin(Waypoint_14_p, qnear=Waypoint_14_q), a=1.3962634015954636, v=1.0471975511965976)
  # begin: URCap Program Node
  #   Source: Robotiq_Grippers, 1.8.11.21258, Robotiq Inc.
  #   Type: Gripper
  $ 360 "Gripper Close (2)"
  if not(gripper_connected[1]):
    popup("Gripper 2 must be connected to run this program.", "No connection", False, True, True)
  end
  if not(rq_is_gripper_activated("2")):
    popup("Gripper 2 is not activated. Go to Installation tab > Gripper to activate it and run the program again.", "Not activated", False, True, True)
  end
  rq_set_pos_spd_for(255, 0, 0, "2")
  rq_wait_pos_spe_for_request(255, 0, 0, "2")
  rq_go_to("2")
  rq_wait("2")
  # end: URCap Program Node
  $ 361 "MoveJ"
  $ 362 "Waypoint_15" "breakAfter"
  movej(get_inverse_kin(Waypoint_15_p, qnear=Waypoint_15_q), a=1.3962634015954636, v=1.0471975511965976)
  $ 363 "MoveJ"
  $ 364 "Waypoint_33" "breakAfter"
  movej(get_inverse_kin(Waypoint_33_p, qnear=Waypoint_33_q), a=1.3962634015954636, v=1.0471975511965976)
  $ 365 "MoveJ"
  $ 366 "Waypoint_34" "breakAfter"
  movej(get_inverse_kin(Waypoint_34_p, qnear=Waypoint_34_q), a=1.3962634015954636, v=1.0471975511965976)
  # begin: URCap Program Node
  #   Source: Robotiq_Grippers, 1.8.11.21258, Robotiq Inc.
  #   Type: Gripper
  $ 367 "Gripper Open (2)"
  if not(gripper_connected[1]):
    popup("Gripper 2 must be connected to run this program.", "No connection", False, True, True)
  end
  if not(rq_is_gripper_activated("2")):
    popup("Gripper 2 is not activated. Go to Installation tab > Gripper to activate it and run the program again.", "Not activated", False, True, True)
  end
  rq_set_pos_spd_for(0, 0, 0, "2")
  rq_wait_pos_spe_for_request(0, 0, 0, "2")
  rq_go_to("2")
  rq_wait("2")
  # end: URCap Program Node
  $ 368 "MoveJ"
  $ 369 "Waypoint_2" "breakAfter"
  movej(get_inverse_kin(Waypoint_2_p, qnear=Waypoint_2_q), a=1.3962634015954636, v=1.0471975511965976)
  $ 370 "MoveJ"
  $ 371 "Waypoint_14" "breakAfter"
  movej(get_inverse_kin(Waypoint_14_p, qnear=Waypoint_14_q), a=1.3962634015954636, v=1.0471975511965976)
  # begin: URCap Program Node
  #   Source: Robotiq_Grippers, 1.8.11.21258, Robotiq Inc.
  #   Type: Gripper
  $ 372 "Gripper Close (2)"
  if not(gripper_connected[1]):
    popup("Gripper 2 must be connected to run this program.", "No connection", False, True, True)
  end
  if not(rq_is_gripper_activated("2")):
    popup("Gripper 2 is not activated. Go to Installation tab > Gripper to activate it and run the program again.", "Not activated", False, True, True)
  end
  rq_set_pos_spd_for(255, 0, 0, "2")
  rq_wait_pos_spe_for_request(255, 0, 0, "2")
  rq_go_to("2")
  rq_wait("2")
  # end: URCap Program Node
  $ 373 "MoveJ"
  $ 374 "Waypoint_15" "breakAfter"
  movej(get_inverse_kin(Waypoint_15_p, qnear=Waypoint_15_q), a=1.3962634015954636, v=1.0471975511965976)
  $ 375 "MoveJ"
  $ 376 "Waypoint_35" "breakAfter"
  movej(get_inverse_kin(Waypoint_35_p, qnear=Waypoint_35_q), a=1.3962634015954636, v=1.0471975511965976)
  $ 377 "MoveJ"
  $ 378 "Waypoint_36" "breakAfter"
  movej(get_inverse_kin(Waypoint_36_p, qnear=Waypoint_36_q), a=1.3962634015954636, v=1.0471975511965976)
  # begin: URCap Program Node
  #   Source: Robotiq_Grippers, 1.8.11.21258, Robotiq Inc.
  #   Type: Gripper
  $ 379 "Gripper Open (2)"
  if not(gripper_connected[1]):
    popup("Gripper 2 must be connected to run this program.", "No connection", False, True, True)
  end
  if not(rq_is_gripper_activated("2")):
    popup("Gripper 2 is not activated. Go to Installation tab > Gripper to activate it and run the program again.", "Not activated", False, True, True)
  end
  rq_set_pos_spd_for(0, 0, 0, "2")
  rq_wait_pos_spe_for_request(0, 0, 0, "2")
  rq_go_to("2")
  rq_wait("2")
  # end: URCap Program Node
  $ 380 "MoveJ"
  $ 381 "Waypoint_37" "breakAfter"
  movej(get_inverse_kin(Waypoint_37_p, qnear=Waypoint_37_q), a=1.3962634015954636, v=1.0471975511965976)
  # begin: URCap Program Node
  #   Source: Robotiq_Grippers, 1.8.11.21258, Robotiq Inc.
  #   Type: Gripper
  $ 382 "Gripper Close (2)"
  if not(gripper_connected[1]):
    popup("Gripper 2 must be connected to run this program.", "No connection", False, True, True)
  end
  if not(rq_is_gripper_activated("2")):
    popup("Gripper 2 is not activated. Go to Installation tab > Gripper to activate it and run the program again.", "Not activated", False, True, True)
  end
  rq_set_pos_spd_for(255, 0, 0, "2")
  rq_wait_pos_spe_for_request(255, 0, 0, "2")
  rq_go_to("2")
  rq_wait("2")
  # end: URCap Program Node
  $ 383 "MoveJ"
  $ 384 "Waypoint_54" "breakAfter"
  movej(get_inverse_kin(Waypoint_54_p, qnear=Waypoint_54_q), a=1.3962634015954636, v=1.0471975511965976)
  # begin: URCap Program Node
  #   Source: Robotiq_Grippers, 1.8.11.21258, Robotiq Inc.
  #   Type: Gripper
  $ 385 "Gripper Open (2)"
  if not(gripper_connected[1]):
    popup("Gripper 2 must be connected to run this program.", "No connection", False, True, True)
  end
  if not(rq_is_gripper_activated("2")):
    popup("Gripper 2 is not activated. Go to Installation tab > Gripper to activate it and run the program again.", "Not activated", False, True, True)
  end
  rq_set_pos_spd_for(0, 0, 0, "2")
  rq_wait_pos_spe_for_request(0, 0, 0, "2")
  rq_go_to("2")
  rq_wait("2")
  # end: URCap Program Node
  $ 386 "MoveJ"
  $ 387 "Waypoint_39" "breakAfter"
  movej(get_inverse_kin(Waypoint_39_p, qnear=Waypoint_39_q), a=1.3962634015954636, v=1.0471975511965976)
  # begin: URCap Program Node
  #   Source: Robotiq_Grippers, 1.8.11.21258, Robotiq Inc.
  #   Type: Gripper
  $ 388 "Gripper Close (2)"
  if not(gripper_connected[1]):
    popup("Gripper 2 must be connected to run this program.", "No connection", False, True, True)
  end
  if not(rq_is_gripper_activated("2")):
    popup("Gripper 2 is not activated. Go to Installation tab > Gripper to activate it and run the program again.", "Not activated", False, True, True)
  end
  rq_set_pos_spd_for(255, 0, 0, "2")
  rq_wait_pos_spe_for_request(255, 0, 0, "2")
  rq_go_to("2")
  rq_wait("2")
  # end: URCap Program Node
  $ 389 "MoveJ"
  $ 390 "Waypoint_40" "breakAfter"
  movej(get_inverse_kin(Waypoint_40_p, qnear=Waypoint_40_q), a=1.3962634015954636, v=1.0471975511965976)
  $ 391 "MoveJ"
  $ 392 "Waypoint_41" "breakAfter"
  movej(get_inverse_kin(Waypoint_41_p, qnear=Waypoint_41_q), a=1.3962634015954636, v=1.0471975511965976)
  $ 393 "MoveJ"
  $ 394 "Waypoint_42" "breakAfter"
  movej(get_inverse_kin(Waypoint_42_p, qnear=Waypoint_42_q), a=1.3962634015954636, v=1.0471975511965976)
  # begin: URCap Program Node
  #   Source: Robotiq_Grippers, 1.8.11.21258, Robotiq Inc.
  #   Type: Gripper
  $ 395 "Gripper Open (2)"
  if not(gripper_connected[1]):
    popup("Gripper 2 must be connected to run this program.", "No connection", False, True, True)
  end
  if not(rq_is_gripper_activated("2")):
    popup("Gripper 2 is not activated. Go to Installation tab > Gripper to activate it and run the program again.", "Not activated", False, True, True)
  end
  rq_set_pos_spd_for(0, 0, 0, "2")
  rq_wait_pos_spe_for_request(0, 0, 0, "2")
  rq_go_to("2")
  rq_wait("2")
  # end: URCap Program Node
  $ 396 "MoveJ"
  $ 397 "Waypoint_55" "breakAfter"
  movej(get_inverse_kin(Waypoint_55_p, qnear=Waypoint_55_q), a=1.3962634015954636, v=1.0471975511965976)
  $ 398 "MoveJ"
  $ 399 "Waypoint_2" "breakAfter"
  movej(get_inverse_kin(Waypoint_2_p, qnear=Waypoint_2_q), a=1.3962634015954636, v=1.0471975511965976)
  $ 400 "MoveJ"
  $ 401 "Waypoint_14" "breakAfter"
  movej(get_inverse_kin(Waypoint_14_p, qnear=Waypoint_14_q), a=1.3962634015954636, v=1.0471975511965976)
  # begin: URCap Program Node
  #   Source: Robotiq_Grippers, 1.8.11.21258, Robotiq Inc.
  #   Type: Gripper
  $ 402 "Gripper Close (2)"
  if not(gripper_connected[1]):
    popup("Gripper 2 must be connected to run this program.", "No connection", False, True, True)
  end
  if not(rq_is_gripper_activated("2")):
    popup("Gripper 2 is not activated. Go to Installation tab > Gripper to activate it and run the program again.", "Not activated", False, True, True)
  end
  rq_set_pos_spd_for(255, 0, 0, "2")
  rq_wait_pos_spe_for_request(255, 0, 0, "2")
  rq_go_to("2")
  rq_wait("2")
  # end: URCap Program Node
  $ 403 "MoveJ"
  $ 404 "Waypoint_43" "breakAfter"
  movej(get_inverse_kin(Waypoint_43_p, qnear=Waypoint_43_q), a=1.3962634015954636, v=1.0471975511965976)
  $ 405 "MoveJ"
  $ 406 "Waypoint_44" "breakAfter"
  movej(get_inverse_kin(Waypoint_44_p, qnear=Waypoint_44_q), a=1.3962634015954636, v=1.0471975511965976)
  $ 407 "MoveJ"
  $ 408 "Waypoint_45" "breakAfter"
  movej(get_inverse_kin(Waypoint_45_p, qnear=Waypoint_45_q), a=1.3962634015954636, v=1.0471975511965976)
  # begin: URCap Program Node
  #   Source: Robotiq_Grippers, 1.8.11.21258, Robotiq Inc.
  #   Type: Gripper
  $ 409 "Gripper Open (2)"
  if not(gripper_connected[1]):
    popup("Gripper 2 must be connected to run this program.", "No connection", False, True, True)
  end
  if not(rq_is_gripper_activated("2")):
    popup("Gripper 2 is not activated. Go to Installation tab > Gripper to activate it and run the program again.", "Not activated", False, True, True)
  end
  rq_set_pos_spd_for(0, 0, 0, "2")
  rq_wait_pos_spe_for_request(0, 0, 0, "2")
  rq_go_to("2")
  rq_wait("2")
  # end: URCap Program Node
  $ 410 "MoveJ"
  $ 411 "Waypoint_2" "breakAfter"
  movej(get_inverse_kin(Waypoint_2_p, qnear=Waypoint_2_q), a=1.3962634015954636, v=1.0471975511965976)
  $ 412 "MoveJ"
  $ 413 "Waypoint_14" "breakAfter"
  movej(get_inverse_kin(Waypoint_14_p, qnear=Waypoint_14_q), a=1.3962634015954636, v=1.0471975511965976)
  # begin: URCap Program Node
  #   Source: Robotiq_Grippers, 1.8.11.21258, Robotiq Inc.
  #   Type: Gripper
  $ 414 "Gripper Close (2)"
  if not(gripper_connected[1]):
    popup("Gripper 2 must be connected to run this program.", "No connection", False, True, True)
  end
  if not(rq_is_gripper_activated("2")):
    popup("Gripper 2 is not activated. Go to Installation tab > Gripper to activate it and run the program again.", "Not activated", False, True, True)
  end
  rq_set_pos_spd_for(255, 0, 0, "2")
  rq_wait_pos_spe_for_request(255, 0, 0, "2")
  rq_go_to("2")
  rq_wait("2")
  # end: URCap Program Node
  $ 415 "MoveJ"
  $ 416 "Waypoint_46" "breakAfter"
  movej(get_inverse_kin(Waypoint_46_p, qnear=Waypoint_46_q), a=1.3962634015954636, v=1.0471975511965976)
  $ 417 "MoveJ"
  $ 418 "Waypoint_47" "breakAfter"
  movej(get_inverse_kin(Waypoint_47_p, qnear=Waypoint_47_q), a=1.3962634015954636, v=1.0471975511965976)
  $ 419 "MoveJ"
  $ 420 "Waypoint_48" "breakAfter"
  movej(get_inverse_kin(Waypoint_48_p, qnear=Waypoint_48_q), a=1.3962634015954636, v=1.0471975511965976)
  # begin: URCap Program Node
  #   Source: Robotiq_Grippers, 1.8.11.21258, Robotiq Inc.
  #   Type: Gripper
  $ 421 "Gripper Open (2)"
  if not(gripper_connected[1]):
    popup("Gripper 2 must be connected to run this program.", "No connection", False, True, True)
  end
  if not(rq_is_gripper_activated("2")):
    popup("Gripper 2 is not activated. Go to Installation tab > Gripper to activate it and run the program again.", "Not activated", False, True, True)
  end
  rq_set_pos_spd_for(0, 0, 0, "2")
  rq_wait_pos_spe_for_request(0, 0, 0, "2")
  rq_go_to("2")
  rq_wait("2")
  # end: URCap Program Node
  $ 422 "MoveJ"
  $ 423 "Waypoint_2" "breakAfter"
  movej(get_inverse_kin(Waypoint_2_p, qnear=Waypoint_2_q), a=1.3962634015954636, v=1.0471975511965976)
  $ 424 "MoveJ"
  $ 425 "Waypoint_52" "breakAfter"
  movej(get_inverse_kin(Waypoint_52_p, qnear=Waypoint_52_q), a=1.3962634015954636, v=1.0471975511965976)
  # begin: URCap Program Node
  #   Source: Robotiq_Grippers, 1.8.11.21258, Robotiq Inc.
  #   Type: Gripper
  $ 426 "Gripper Close (2)"
  if not(gripper_connected[1]):
    popup("Gripper 2 must be connected to run this program.", "No connection", False, True, True)
  end
  if not(rq_is_gripper_activated("2")):
    popup("Gripper 2 is not activated. Go to Installation tab > Gripper to activate it and run the program again.", "Not activated", False, True, True)
  end
  rq_set_pos_spd_for(255, 0, 0, "2")
  rq_wait_pos_spe_for_request(255, 0, 0, "2")
  rq_go_to("2")
  rq_wait("2")
  # end: URCap Program Node
  $ 427 "MoveJ"
  $ 428 "Waypoint_49" "breakAfter"
  movej(get_inverse_kin(Waypoint_49_p, qnear=Waypoint_49_q), a=1.3962634015954636, v=1.0471975511965976)
  $ 429 "MoveJ"
  $ 430 "Waypoint_50" "breakAfter"
  movej(get_inverse_kin(Waypoint_50_p, qnear=Waypoint_50_q), a=1.3962634015954636, v=1.0471975511965976)
  # begin: URCap Program Node
  #   Source: Robotiq_Grippers, 1.8.11.21258, Robotiq Inc.
  #   Type: Gripper
  $ 431 "Gripper Open (2)"
  if not(gripper_connected[1]):
    popup("Gripper 2 must be connected to run this program.", "No connection", False, True, True)
  end
  if not(rq_is_gripper_activated("2")):
    popup("Gripper 2 is not activated. Go to Installation tab > Gripper to activate it and run the program again.", "Not activated", False, True, True)
  end
  rq_set_pos_spd_for(0, 0, 0, "2")
  rq_wait_pos_spe_for_request(0, 0, 0, "2")
  rq_go_to("2")
  rq_wait("2")
  # end: URCap Program Node
  $ 432 "MoveJ"
  $ 433 "Waypoint_2" "breakAfter"
  movej(get_inverse_kin(Waypoint_2_p, qnear=Waypoint_2_q), a=1.3962634015954636, v=1.0471975511965976)
  $ 434 "MoveJ"
  $ 435 "Waypoint_14" "breakAfter"
  movej(get_inverse_kin(Waypoint_14_p, qnear=Waypoint_14_q), a=1.3962634015954636, v=1.0471975511965976)
  # begin: URCap Program Node
  #   Source: Robotiq_Grippers, 1.8.11.21258, Robotiq Inc.
  #   Type: Gripper
  $ 436 "Gripper Close (2)"
  if not(gripper_connected[1]):
    popup("Gripper 2 must be connected to run this program.", "No connection", False, True, True)
  end
  if not(rq_is_gripper_activated("2")):
    popup("Gripper 2 is not activated. Go to Installation tab > Gripper to activate it and run the program again.", "Not activated", False, True, True)
  end
  rq_set_pos_spd_for(255, 0, 0, "2")
  rq_wait_pos_spe_for_request(255, 0, 0, "2")
  rq_go_to("2")
  rq_wait("2")
  # end: URCap Program Node
  $ 437 "MoveJ"
  $ 438 "Waypoint_51" "breakAfter"
  movej(get_inverse_kin(Waypoint_51_p, qnear=Waypoint_51_q), a=1.3962634015954636, v=1.0471975511965976)
  $ 439 "MoveJ"
  $ 440 "Waypoint_53" "breakAfter"
  movej(get_inverse_kin(Waypoint_53_p, qnear=Waypoint_53_q), a=1.3962634015954636, v=1.0471975511965976)
  # begin: URCap Program Node
  #   Source: Robotiq_Grippers, 1.8.11.21258, Robotiq Inc.
  #   Type: Gripper
  $ 441 "Gripper Open (2)"
  if not(gripper_connected[1]):
    popup("Gripper 2 must be connected to run this program.", "No connection", False, True, True)
  end
  if not(rq_is_gripper_activated("2")):
    popup("Gripper 2 is not activated. Go to Installation tab > Gripper to activate it and run the program again.", "Not activated", False, True, True)
  end
  rq_set_pos_spd_for(0, 0, 0, "2")
  rq_wait_pos_spe_for_request(0, 0, 0, "2")
  rq_go_to("2")
  rq_wait("2")
  # end: URCap Program Node
  $ 442 "MoveJ"
  $ 443 "Waypoint_2" "breakAfter"
  movej(get_inverse_kin(Waypoint_2_p, qnear=Waypoint_2_q), a=1.3962634015954636, v=1.0471975511965976)
  $ 444 "Mouvement D"
  $ 445 "MoveJ"
  $ 446 "Waypoint_2" "breakAfter"
  movej(get_inverse_kin(Waypoint_2_p, qnear=Waypoint_2_q), a=1.3962634015954636, v=1.0471975511965976)
  $ 447 "MoveJ"
  $ 448 "Waypoint_56" "breakAfter"
  movej(get_inverse_kin(Waypoint_56_p, qnear=Waypoint_56_q), a=1.3962634015954636, v=1.0471975511965976)
  # begin: URCap Program Node
  #   Source: Robotiq_Grippers, 1.8.11.21258, Robotiq Inc.
  #   Type: Gripper
  $ 449 "Gripper Close (2)"
  if not(gripper_connected[1]):
    popup("Gripper 2 must be connected to run this program.", "No connection", False, True, True)
  end
  if not(rq_is_gripper_activated("2")):
    popup("Gripper 2 is not activated. Go to Installation tab > Gripper to activate it and run the program again.", "Not activated", False, True, True)
  end
  rq_set_pos_spd_for(255, 0, 0, "2")
  rq_wait_pos_spe_for_request(255, 0, 0, "2")
  rq_go_to("2")
  rq_wait("2")
  # end: URCap Program Node
  $ 450 "MoveJ"
  $ 451 "Waypoint_57" "breakAfter"
  movej(get_inverse_kin(Waypoint_57_p, qnear=Waypoint_57_q), a=1.3962634015954636, v=1.0471975511965976)
  $ 452 "MoveJ"
  $ 453 "Waypoint_58" "breakAfter"
  movej(get_inverse_kin(Waypoint_58_p, qnear=Waypoint_58_q), a=1.3962634015954636, v=1.0471975511965976)
  # begin: URCap Program Node
  #   Source: Robotiq_Grippers, 1.8.11.21258, Robotiq Inc.
  #   Type: Gripper
  $ 454 "Gripper Open (2)"
  if not(gripper_connected[1]):
    popup("Gripper 2 must be connected to run this program.", "No connection", False, True, True)
  end
  if not(rq_is_gripper_activated("2")):
    popup("Gripper 2 is not activated. Go to Installation tab > Gripper to activate it and run the program again.", "Not activated", False, True, True)
  end
  rq_set_pos_spd_for(0, 0, 0, "2")
  rq_wait_pos_spe_for_request(0, 0, 0, "2")
  rq_go_to("2")
  rq_wait("2")
  # end: URCap Program Node
  $ 455 "MoveJ"
  $ 456 "Waypoint_2" "breakAfter"
  movej(get_inverse_kin(Waypoint_2_p, qnear=Waypoint_2_q), a=1.3962634015954636, v=1.0471975511965976)
  $ 457 "MoveJ"
  $ 458 "Waypoint_56" "breakAfter"
  movej(get_inverse_kin(Waypoint_56_p, qnear=Waypoint_56_q), a=1.3962634015954636, v=1.0471975511965976)
  # begin: URCap Program Node
  #   Source: Robotiq_Grippers, 1.8.11.21258, Robotiq Inc.
  #   Type: Gripper
  $ 459 "Gripper Close (2)"
  if not(gripper_connected[1]):
    popup("Gripper 2 must be connected to run this program.", "No connection", False, True, True)
  end
  if not(rq_is_gripper_activated("2")):
    popup("Gripper 2 is not activated. Go to Installation tab > Gripper to activate it and run the program again.", "Not activated", False, True, True)
  end
  rq_set_pos_spd_for(255, 0, 0, "2")
  rq_wait_pos_spe_for_request(255, 0, 0, "2")
  rq_go_to("2")
  rq_wait("2")
  # end: URCap Program Node
  $ 460 "MoveJ"
  $ 461 "Waypoint_57" "breakAfter"
  movej(get_inverse_kin(Waypoint_57_p, qnear=Waypoint_57_q), a=1.3962634015954636, v=1.0471975511965976)
  $ 462 "MoveJ"
  $ 463 "Waypoint_58" "breakAfter"
  movej(get_inverse_kin(Waypoint_58_p, qnear=Waypoint_58_q), a=1.3962634015954636, v=1.0471975511965976)
  # begin: URCap Program Node
  #   Source: Robotiq_Grippers, 1.8.11.21258, Robotiq Inc.
  #   Type: Gripper
  $ 464 "Gripper Open (2)"
  if not(gripper_connected[1]):
    popup("Gripper 2 must be connected to run this program.", "No connection", False, True, True)
  end
  if not(rq_is_gripper_activated("2")):
    popup("Gripper 2 is not activated. Go to Installation tab > Gripper to activate it and run the program again.", "Not activated", False, True, True)
  end
  rq_set_pos_spd_for(0, 0, 0, "2")
  rq_wait_pos_spe_for_request(0, 0, 0, "2")
  rq_go_to("2")
  rq_wait("2")
  # end: URCap Program Node
  $ 465 "MoveJ"
  $ 466 "Waypoint_2" "breakAfter"
  movej(get_inverse_kin(Waypoint_2_p, qnear=Waypoint_2_q), a=1.3962634015954636, v=1.0471975511965976)
  $ 467 "MoveJ"
  $ 468 "Waypoint_59" "breakAfter"
  movej(get_inverse_kin(Waypoint_59_p, qnear=Waypoint_59_q), a=1.3962634015954636, v=1.0471975511965976)
  # begin: URCap Program Node
  #   Source: Robotiq_Grippers, 1.8.11.21258, Robotiq Inc.
  #   Type: Gripper
  $ 469 "Gripper Close (2)"
  if not(gripper_connected[1]):
    popup("Gripper 2 must be connected to run this program.", "No connection", False, True, True)
  end
  if not(rq_is_gripper_activated("2")):
    popup("Gripper 2 is not activated. Go to Installation tab > Gripper to activate it and run the program again.", "Not activated", False, True, True)
  end
  rq_set_pos_spd_for(255, 0, 0, "2")
  rq_wait_pos_spe_for_request(255, 0, 0, "2")
  rq_go_to("2")
  rq_wait("2")
  # end: URCap Program Node
  $ 470 "MoveJ"
  $ 471 "Waypoint_60" "breakAfter"
  movej(get_inverse_kin(Waypoint_60_p, qnear=Waypoint_60_q), a=1.3962634015954636, v=1.0471975511965976)
  # begin: URCap Program Node
  #   Source: Robotiq_Grippers, 1.8.11.21258, Robotiq Inc.
  #   Type: Gripper
  $ 472 "Gripper Open (2)"
  if not(gripper_connected[1]):
    popup("Gripper 2 must be connected to run this program.", "No connection", False, True, True)
  end
  if not(rq_is_gripper_activated("2")):
    popup("Gripper 2 is not activated. Go to Installation tab > Gripper to activate it and run the program again.", "Not activated", False, True, True)
  end
  rq_set_pos_spd_for(0, 0, 0, "2")
  rq_wait_pos_spe_for_request(0, 0, 0, "2")
  rq_go_to("2")
  rq_wait("2")
  # end: URCap Program Node
  $ 473 "MoveJ"
  $ 474 "Waypoint_2" "breakAfter"
  movej(get_inverse_kin(Waypoint_2_p, qnear=Waypoint_2_q), a=1.3962634015954636, v=1.0471975511965976)
  $ 475 "MoveJ"
  $ 476 "Waypoint_2" "breakAfter"
  movej(get_inverse_kin(Waypoint_2_p, qnear=Waypoint_2_q), a=1.3962634015954636, v=1.0471975511965976)
  $ 477 "MoveJ"
  $ 478 "Waypoint_56" "breakAfter"
  movej(get_inverse_kin(Waypoint_56_p, qnear=Waypoint_56_q), a=1.3962634015954636, v=1.0471975511965976)
  # begin: URCap Program Node
  #   Source: Robotiq_Grippers, 1.8.11.21258, Robotiq Inc.
  #   Type: Gripper
  $ 479 "Gripper Close (2)"
  if not(gripper_connected[1]):
    popup("Gripper 2 must be connected to run this program.", "No connection", False, True, True)
  end
  if not(rq_is_gripper_activated("2")):
    popup("Gripper 2 is not activated. Go to Installation tab > Gripper to activate it and run the program again.", "Not activated", False, True, True)
  end
  rq_set_pos_spd_for(255, 0, 0, "2")
  rq_wait_pos_spe_for_request(255, 0, 0, "2")
  rq_go_to("2")
  rq_wait("2")
  # end: URCap Program Node
  $ 480 "MoveJ"
  $ 481 "Waypoint_57" "breakAfter"
  movej(get_inverse_kin(Waypoint_57_p, qnear=Waypoint_57_q), a=1.3962634015954636, v=1.0471975511965976)
  $ 482 "MoveJ"
  $ 483 "Waypoint_58" "breakAfter"
  movej(get_inverse_kin(Waypoint_58_p, qnear=Waypoint_58_q), a=1.3962634015954636, v=1.0471975511965976)
  # begin: URCap Program Node
  #   Source: Robotiq_Grippers, 1.8.11.21258, Robotiq Inc.
  #   Type: Gripper
  $ 484 "Gripper Open (2)"
  if not(gripper_connected[1]):
    popup("Gripper 2 must be connected to run this program.", "No connection", False, True, True)
  end
  if not(rq_is_gripper_activated("2")):
